Yaskawa INFORM job: CPRINT3D.JBI

/JOB
//NAME CPRINT3D
//POS
///NPOS 981,0,0,0,0,0
///TOOL 9
///POSTYPE PULSE
///PULSE
C00000=20899,58707,-95028,75516,-125126,-84020,0
C00001=20890,61280,-94031,74948,-124335,-84934,0
C00002=20888,61868,-93778,74829,-124164,-85130,0
C00003=21010,62075,-93213,74809,-124380,-84988,0
C00004=21199,62234,-92779,74700,-124608,-84895,0
C00005=21337,62300,-92602,74597,-124739,-84867,0
C00006=38851,62476,-92387,77627,-123060,-84391,0
C00007=39075,62591,-92079,77464,-123273,-84335,0
C00008=39325,62631,-91976,77240,-123458,-84342,0
C00009=39575,62590,-92092,76980,-123593,-84413,0
C00010=39796,62473,-92413,76711,-123659,-84538,0
C00011=39905,62372,-92691,76558,-123665,-84634,0
C00012=51767,54029,-117549,60022,-121835,-93519,0
C00013=51973,53909,-117950,59735,-121747,-93661,0
C00014=52088,53762,-118443,59535,-121588,-93813,0
C00015=52099,53603,-118972,59445,-121375,-93959,0
C00016=52003,53453,-119474,59478,-121135,-94082,0
C00017=51897,53373,-119741,59558,-120988,-94140,0
C00018=29408,51344,-126354,60860,-117429,-95669,0
C00019=29082,51299,-126517,61201,-117262,-95677,0
C00020=28737,51300,-126508,61583,-117162,-95633,0
C00021=28416,51346,-126329,61959,-117138,-95543,0
C00022=28156,51432,-126000,62285,-117193,-95416,0
C00023=28041,51501,-125745,62442,-117261,-95327,0
C00024=20896,61411,-95034,74604,-123854,-85488,0
C00025=20848,61637,-94410,74758,-123981,-85303,0
C00026=20875,61793,-93981,74806,-124105,-85185,0
C00027=23614,61599,-94547,71990,-125641,-85793,0
C00028=23696,61485,-94861,71849,-125604,-85896,0
C00029=23753,61360,-95207,71729,-125543,-86002,0
C00030=23779,61231,-95564,71637,-125461,-86108,0
C00031=23776,61103,-95917,71576,-125361,-86206,0
C00032=23744,60981,-96255,71547,-125249,-86296,0
C00033=23690,60879,-96538,71550,-125138,-86366,0
C00034=23633,60785,-96800,71560,-125033,-86431,0
C00035=23546,60693,-97055,71602,-124911,-86488,0
C00036=23440,60617,-97265,71672,-124790,-86529,0
C00037=23318,60561,-97421,71767,-124676,-86553,0
C00038=23186,60525,-97517,71884,-124572,-86559,0
C00039=23047,60513,-97550,72018,-124482,-86545,0
C00040=22909,60524,-97518,72163,-124411,-86514,0
C00041=22788,60555,-97430,72301,-124363,-86469,0
C00042=22668,60592,-97325,72440,-124321,-86420,0
C00043=22545,60656,-97145,72595,-124297,-86349,0
C00044=22438,60742,-96904,72745,-124300,-86264,0
C00045=22352,60847,-96612,72882,-124326,-86167,0
C00046=22291,60967,-96277,73001,-124380,-86062,0
C00047=22259,61099,-95912,73098,-124457,-85954,0
C00048=22258,61236,-95531,73166,-124557,-85845,0
C00049=22288,61375,-95148,73204,-124675,-85742,0
C00050=22350,61509,-94780,73208,-124810,-85648,0
C00051=22446,61639,-94424,73177,-124961,-85563,0
C00052=22581,61738,-94153,73092,-125115,-85509,0
C00053=22727,61808,-93962,72982,-125256,-85479,0
C00054=22884,61852,-93844,72847,-125383,-85472,0
C00055=23056,61868,-93803,72683,-125500,-85489,0
C00056=23225,61837,-93889,72500,-125581,-85542,0
C00057=23374,61780,-94048,72322,-125629,-85611,0
C00058=23505,61699,-94271,72150,-125649,-85697,0
C00059=23556,61652,-94401,72074,-125645,-85742,0
C00060=23536,61543,-94699,72039,-125552,-85823,0
C00061=23608,61444,-94973,71917,-125521,-85912,0
C00062=23657,61335,-95274,71813,-125468,-86005,0
C00063=23680,61224,-95582,71734,-125397,-86095,0
C00064=23677,61113,-95888,71681,-125311,-86181,0
C00065=23649,61009,-96178,71656,-125214,-86258,0
C00066=23600,60916,-96433,71659,-125115,-86322,0
C00067=23549,60831,-96669,71669,-125019,-86380,0
C00068=23474,60752,-96888,71705,-124914,-86429,0
C00069=23383,60687,-97068,71764,-124812,-86464,0
C00070=23279,60639,-97201,71846,-124713,-86485,0
C00071=23166,60609,-97284,71946,-124625,-86489,0
C00072=23048,60598,-97312,72060,-124548,-86478,0
C00073=22929,60608,-97284,72184,-124486,-86451,0
C00074=22820,60636,-97205,72308,-124443,-86410,0
C00075=22712,60669,-97111,72433,-124405,-86366,0
C00076=22606,60724,-96956,72566,-124385,-86305,0
C00077=22514,60798,-96748,72696,-124386,-86232,0
C00078=22440,60889,-96494,72815,-124410,-86148,0
C00079=22387,60994,-96204,72919,-124456,-86057,0
C00080=22359,61109,-95885,73003,-124524,-85962,0
C00081=22357,61229,-95552,73063,-124611,-85868,0
C00082=22384,61351,-95217,73097,-124716,-85777,0
C00083=22437,61468,-94894,73101,-124833,-85694,0
C00084=22520,61579,-94589,73074,-124964,-85622,0
C00085=22635,61664,-94357,73001,-125095,-85575,0
C00086=22764,61725,-94189,72903,-125219,-85549,0
C00087=22903,61764,-94085,72784,-125332,-85543,0
C00088=23051,61778,-94049,72643,-125431,-85557,0
C00089=23195,61751,-94124,72486,-125499,-85603,0
C00090=23326,61701,-94262,72330,-125542,-85664,0
C00091=23441,61631,-94458,72179,-125559,-85738,0
C00092=23479,61596,-94553,72124,-125557,-85772,0
C00093=23667,61562,-94650,71917,-125644,-85831,0
C00094=22262,61550,-94666,73316,-124787,-85601,0
C00095=22193,61400,-95079,73311,-124636,-85707,0
C00096=22159,61244,-95509,73269,-124503,-85823,0
C00097=22160,61140,-95796,73217,-124427,-85904,0
C00098=22111,61132,-95819,73262,-124393,-85903,0
C00099=21934,61528,-94723,73632,-124571,-85564,0
C00100=22292,61657,-94372,73339,-124881,-85523,0
C00101=22319,61626,-94456,73297,-124876,-85551,0
C00102=22308,61612,-94496,73300,-124859,-85560,0
C00103=29023,52904,-120775,62001,-119581,-94025,0
C00104=29186,52950,-120622,61843,-119699,-94004,0
C00105=29368,52980,-120522,61657,-119804,-94001,0
C00106=29561,52993,-120481,61451,-119889,-94017,0
C00107=29759,52988,-120500,61230,-119951,-94051,0
C00108=29955,52965,-120584,61003,-119987,-94102,0
C00109=30150,52921,-120738,60768,-119993,-94173,0
C00110=30308,52852,-120980,60560,-119950,-94263,0
C00111=30428,52773,-121251,60391,-119880,-94355,0
C00112=30513,52686,-121554,60255,-119785,-94452,0
C00113=30562,52588,-121893,60155,-119660,-94553,0
C00114=30545,52489,-122240,60127,-119511,-94648,0
C00115=30488,52400,-122551,60150,-119363,-94727,0
C00116=30393,52319,-122833,60217,-119215,-94794,0
C00117=30266,52250,-123075,60325,-119072,-94844,0
C00118=30114,52195,-123269,60468,-118942,-94878,0
C00119=29942,52155,-123408,60639,-118828,-94894,0
C00120=29759,52131,-123489,60831,-118734,-94894,0
C00121=29572,52123,-123512,61034,-118664,-94875,0
C00122=29390,52132,-123478,61239,-118619,-94842,0
C00123=29234,52154,-123395,61422,-118601,-94798,0
C00124=29088,52179,-123303,61594,-118591,-94752,0
C00125=28943,52220,-123155,61773,-118602,-94691,0
C00126=28819,52274,-122964,61934,-118638,-94621,0
C00127=28723,52337,-122739,62069,-118695,-94543,0
C00128=28656,52408,-122490,62175,-118773,-94463,0
C00129=28623,52483,-122223,62246,-118868,-94383,0
C00130=28624,52561,-121951,62282,-118976,-94305,0
C00131=28655,52632,-121706,62280,-119085,-94239,0
C00132=28695,52703,-121461,62269,-119195,-94175,0
C00133=28773,52778,-121205,62217,-119324,-94113,0
C00134=28884,52846,-120972,62127,-119455,-94062,0
C00135=28945,52871,-120885,62072,-119510,-94046,0
C00136=29095,52857,-120937,61900,-119543,-94081,0
C00137=29237,52897,-120804,61762,-119645,-94063,0
C00138=29396,52923,-120718,61600,-119736,-94061,0
C00139=29565,52935,-120681,61419,-119811,-94074,0
C00140=29739,52930,-120698,61225,-119865,-94104,0
C00141=29911,52910,-120772,61025,-119896,-94148,0
C00142=30078,52872,-120904,60823,-119901,-94209,0
C00143=30214,52813,-121110,60646,-119864,-94286,0
C00144=30320,52744,-121350,60497,-119802,-94368,0
C00145=30395,52667,-121617,60378,-119718,-94453,0
C00146=30436,52584,-121908,60292,-119612,-94540,0
C00147=30421,52498,-122205,60269,-119485,-94621,0
C00148=30370,52420,-122477,60289,-119355,-94690,0
C00149=30287,52350,-122724,60348,-119225,-94748,0
C00150=30176,52289,-122936,60442,-119101,-94793,0
C00151=30043,52241,-123104,60567,-118987,-94823,0
C00152=29894,52206,-123225,60715,-118888,-94836,0
C00153=29736,52185,-123296,60881,-118807,-94836,0
C00154=29575,52179,-123316,61056,-118746,-94820,0
C00155=29419,52186,-123286,61232,-118707,-94791,0
C00156=29279,52206,-123211,61396,-118691,-94751,0
C00157=29148,52229,-123130,61551,-118681,-94711,0
C00158=29023,52264,-123002,61705,-118691,-94658,0
C00159=28917,52310,-122839,61843,-118722,-94597,0
C00160=28834,52364,-122646,61959,-118771,-94532,0
C00161=28777,52425,-122432,62050,-118838,-94463,0
C00162=28749,52490,-122204,62111,-118918,-94394,0
C00163=28749,52556,-121970,62142,-119011,-94328,0
C00164=28777,52620,-121750,62141,-119109,-94268,0
C00165=28812,52684,-121530,62131,-119209,-94210,0
C00166=28879,52748,-121308,62087,-119319,-94157,0
C00167=28975,52807,-121107,62009,-119433,-94113,0
C00168=29017,52824,-121047,61971,-119472,-94101,0
C00169=29079,52934,-120675,61954,-119641,-94004,0
C00170=48817,53183,-120295,62872,-119678,-93851,0
C00171=48657,53224,-120148,63068,-119677,-93787,0
C00172=48515,53282,-119949,63250,-119702,-93711,0
C00173=48399,53354,-119702,63411,-119755,-93624,0
C00174=48315,53438,-119417,63544,-119832,-93531,0
C00175=48265,53531,-119102,63641,-119933,-93435,0
C00176=48255,53630,-118772,63700,-120053,-93339,0
C00177=48286,53736,-118420,63715,-120197,-93244,0
C00178=48378,53834,-118099,63660,-120352,-93165,0
C00179=48500,53917,-117828,63567,-120500,-93106,0
C00180=48649,53987,-117600,63436,-120643,-93063,0
C00181=48830,54045,-117416,63265,-120782,-93038,0
C00182=49033,54072,-117332,63055,-120891,-93043,0
C00183=49230,54078,-117320,62842,-120972,-93069,0
C00184=49421,54063,-117371,62626,-121026,-93112,0
C00185=49598,54031,-117484,62415,-121050,-93170,0
C00186=49755,53982,-117647,62219,-121046,-93239,0
C00187=49891,53919,-117860,62040,-121015,-93318,0
C00188=49996,53845,-118106,61888,-120959,-93403,0
C00189=50069,53764,-118377,61769,-120880,-93490,0
C00190=50108,53679,-118661,61685,-120783,-93574,0
C00191=50111,53600,-118923,61643,-120681,-93648,0
C00192=50107,53526,-119172,61613,-120581,-93717,0
C00193=50069,53445,-119442,61616,-120461,-93787,0
C00194=50000,53370,-119695,61656,-120336,-93848,0
C00195=49902,53303,-119919,61733,-120212,-93897,0
C00196=49778,53246,-120107,61842,-120094,-93933,0
C00197=49634,53202,-120252,61980,-119986,-93953,0
C00198=49475,53172,-120349,62141,-119891,-93958,0
C00199=49321,53160,-120388,62305,-119821,-93947,0
C00200=49166,53151,-120413,62473,-119756,-93933,0
C00201=48989,53158,-120383,62670,-119705,-93900,0
C00202=48915,53169,-120345,62757,-119694,-93879,0
C00203=48866,53237,-120111,62843,-119767,-93806,0
C00204=48727,53273,-119983,63013,-119766,-93750,0
C00205=48605,53324,-119811,63171,-119788,-93684,0
C00206=48504,53387,-119595,63312,-119833,-93609,0
C00207=48429,53460,-119346,63428,-119901,-93527,0
C00208=48386,53542,-119071,63514,-119989,-93443,0
C00209=48376,53628,-118781,63566,-120095,-93359,0
C00210=48402,53719,-118480,63580,-120219,-93277,0
C00211=48481,53803,-118204,63533,-120352,-93210,0
C00212=48588,53876,-117964,63450,-120483,-93157,0
C00213=48720,53938,-117764,63335,-120608,-93119,0
C00214=48875,53987,-117607,63188,-120728,-93097,0
C00215=49050,54010,-117534,63008,-120821,-93103,0
C00216=49223,54015,-117524,62820,-120891,-93125,0
C00217=49390,54003,-117569,62631,-120938,-93163,0
C00218=49546,53975,-117667,62446,-120959,-93213,0
C00219=49683,53932,-117810,62275,-120956,-93274,0
C00220=49800,53877,-117994,62119,-120929,-93343,0
C00221=49891,53814,-118208,61988,-120880,-93416,0
C00222=49954,53744,-118442,61886,-120812,-93491,0
C00223=49987,53670,-118686,61814,-120728,-93564,0
C00224=49990,53600,-118923,61777,-120637,-93630,0
C00225=49986,53533,-119147,61750,-120548,-93693,0
C00226=49953,53463,-119378,61753,-120444,-93753,0
C00227=49894,53399,-119594,61787,-120337,-93805,0
C00228=49809,53341,-119787,61853,-120232,-93847,0
C00229=49704,53292,-119948,61946,-120130,-93877,0
C00230=49580,53255,-120072,62064,-120037,-93895,0
C00231=49444,53229,-120155,62202,-119957,-93899,0
C00232=49306,53218,-120190,62350,-119894,-93889,0
C00233=49166,53210,-120212,62500,-119835,-93876,0
C00234=49015,53216,-120187,62670,-119790,-93848,0
C00235=48964,53223,-120161,62728,-119782,-93834,0
C00236=48738,53191,-120265,62963,-119662,-93832,0
C00237=49561,53062,-120729,61994,-119772,-94078,0
C00238=30717,52351,-122728,59873,-119365,-94808,0
C00239=30793,52470,-122309,59844,-119565,-94702,0
C00240=30814,52599,-121862,59881,-119758,-94580,0
C00241=30750,52724,-121427,60011,-119918,-94449,0
C00242=30644,52832,-121052,60179,-120036,-94330,0
C00243=30495,52929,-120716,60390,-120122,-94216,0
C00244=30292,53019,-120407,60657,-120176,-94101,0
C00245=30041,53076,-120209,60960,-120168,-94009,0
C00246=29799,53105,-120105,61241,-120124,-93946,0
C00247=29553,53111,-120080,61515,-120045,-93903,0
C00248=29312,53094,-120133,61773,-119939,-93884,0
C00249=29084,53056,-120258,62005,-119808,-93887,0
C00250=28879,52998,-120450,62204,-119658,-93913,0
C00251=28702,52924,-120699,62363,-119497,-93960,0
C00252=28562,52837,-120996,62478,-119331,-94024,0
C00253=28461,52742,-121323,62544,-119166,-94104,0
C00254=28412,52657,-121616,62558,-119034,-94181,0
C00255=28369,52561,-121948,62562,-118889,-94270,0
C00256=22538,60451,-97717,72502,-124139,-86510,0
C00257=22723,60394,-97878,72288,-124203,-86586,0
C00258=22869,60358,-97983,72122,-124259,-86639,0
C00259=23047,60344,-98024,71935,-124352,-86680,0
C00260=23226,60359,-97982,71762,-124467,-86696,0
C00261=23396,60404,-97858,71611,-124601,-86690,0
C00262=23553,60477,-97658,71487,-124747,-86659,0
C00263=23690,60574,-97388,71397,-124902,-86606,0
C00264=23801,60692,-97061,71343,-125058,-86532,0
C00265=23870,60805,-96746,71330,-125187,-86456,0
C00266=23934,60927,-96407,71327,-125319,-86371,0
C00267=23974,61083,-95975,71365,-125463,-86256,0
C00268=23978,61246,-95525,71444,-125590,-86130,0
C00269=23944,61410,-95073,71561,-125695,-85997,0
C00270=23873,61568,-94637,71714,-125772,-85863,0
C00271=23768,61711,-94241,71892,-125816,-85733,0
C00272=23632,61836,-93895,72092,-125828,-85613,0
C00273=23468,61937,-93617,72307,-125803,-85506,0
C00274=23380,61971,-93523,72413,-125774,-85465,0
C00275=38247,60799,-96991,77469,-121636,-85632,0
C00276=38229,60634,-97453,77414,-121520,-85763,0
C00277=38224,60505,-97812,77364,-121434,-85867,0
C00278=38252,60358,-98224,77272,-121355,-85990,0
C00279=38315,60220,-98614,77149,-121301,-86112,0
C00280=38410,60095,-98966,77001,-121276,-86226,0
C00281=38534,59989,-99267,76833,-121277,-86331,0
C00282=38681,59906,-99506,76650,-121307,-86420,0
C00283=38846,59848,-99673,76460,-121365,-86492,0
C00284=38995,59822,-99749,76300,-121432,-86534,0
C00285=39152,59803,-99808,76134,-121511,-86573,0
C00286=39341,59810,-99789,75949,-121624,-86594,0
C00287=39527,59849,-99684,75780,-121759,-86589,0
C00288=39702,59918,-99492,75635,-121908,-86558,0
C00289=39859,60016,-99219,75522,-122067,-86502,0
C00290=39990,60139,-98875,75446,-122229,-86422,0
C00291=40090,60284,-98470,75413,-122389,-86319,0
C00292=40154,60445,-98019,75422,-122538,-86199,0
C00293=40165,60527,-97789,75448,-122601,-86135,0
C00294=49264,54203,-116909,62865,-121141,-92959,0
C00295=49001,54196,-116927,63150,-121033,-92924,0
C00296=48740,54161,-117035,63420,-120891,-92916,0
C00297=48507,54087,-117270,63639,-120712,-92949,0
C00298=48323,53999,-117551,63799,-120536,-93002,0
C00299=48172,53896,-117887,63915,-120353,-93075,0
C00300=48053,53770,-118301,63986,-120153,-93176,0
C00301=48012,53634,-118754,63967,-119970,-93300,0
C00302=48024,53511,-119164,63896,-119820,-93419,0
C00303=48085,53395,-119556,63776,-119695,-93540,0
C00304=48190,53290,-119913,63611,-119597,-93656,0
C00305=48335,53199,-120225,63409,-119532,-93765,0
C00306=48514,53127,-120476,63179,-119500,-93862,0
C00307=48718,53074,-120661,62930,-119501,-93942,0
C00308=48938,53043,-120775,62673,-119534,-94005,0
C00309=49164,53034,-120813,62419,-119600,-94047,0
C00310=49352,53044,-120783,62217,-119677,-94064,0
C00311=49459,53053,-120756,62103,-119725,-94071,0
C00312=50348,53502,-119261,61335,-120633,-93777,0
C00313=50354,53603,-118923,61377,-120769,-93684,0
C00314=50347,53723,-118523,61442,-120924,-93571,0
C00315=50567,53630,-118838,61154,-120880,-93692,0
C00316=50415,53540,-119133,61280,-120708,-93751,0
C00317=29384,52018,-123887,61194,-118449,-94958,0
C00318=29114,51954,-124111,61462,-118270,-94987,0
C00319=28946,52085,-123636,61708,-118408,-94829,0
C00320=29144,52051,-123761,61474,-118423,-94890,0
C00321=29282,52032,-123833,61312,-118438,-94929,0
C00322=28535,52391,-122546,62301,-118709,-94463,0
C00323=28611,52310,-122832,62180,-118620,-94556,0
C00324=28721,52238,-123089,62026,-118555,-94643,0
C00325=28862,52177,-123307,61842,-118514,-94724,0
C00326=29028,52130,-123477,61638,-118500,-94795,0
C00327=29189,52103,-123578,61448,-118511,-94844,0
C00328=29361,52078,-123669,61246,-118531,-94892,0
C00329=29569,52068,-123709,61012,-118583,-94931,0
C00330=29760,52076,-123686,60804,-118654,-94950,0
C00331=29778,52051,-123776,60773,-118623,-94977,0
C00332=29062,51880,-124374,61486,-118145,-95056,0
C00333=22333,60653,-97151,72807,-124171,-86316,0
C00334=22373,60676,-97086,72778,-124212,-86305,0
C00335=22483,60588,-97333,72624,-124210,-86392,0
C00336=22623,60515,-97539,72447,-124238,-86474,0
C00337=22755,60475,-97654,72294,-124283,-86527,0
C00338=22889,60441,-97751,72142,-124335,-86576,0
C00339=23047,60428,-97787,71976,-124417,-86612,0
C00340=23206,60442,-97750,71823,-124519,-86628,0
C00341=23357,60482,-97640,71689,-124639,-86622,0
C00342=23497,60547,-97462,71580,-124768,-86594,0
C00343=23618,60633,-97222,71500,-124906,-86547,0
C00344=23717,60738,-96931,71452,-125045,-86481,0
C00345=23780,60842,-96642,71440,-125163,-86411,0
C00346=23839,60954,-96331,71437,-125284,-86333,0
C00347=23875,61093,-95946,71470,-125412,-86231,0
C00348=23878,61238,-95544,71540,-125526,-86119,0
C00349=23848,61385,-95140,71645,-125619,-86000,0
C00350=23785,61526,-94749,71781,-125688,-85879,0
C00351=23691,61655,-94394,71941,-125728,-85763,0
C00352=23568,61768,-94083,72121,-125738,-85655,0
C00353=23421,61858,-93832,72314,-125716,-85559,0
C00354=23254,61923,-93655,72514,-125661,-85481,0
C00355=23157,61940,-93605,72620,-125614,-85450,0
C00356=23152,61980,-93497,72644,-125641,-85419,0
C00357=38423,61024,-96369,77395,-121886,-85476,0
C00358=38460,60998,-96443,77347,-121892,-85503,0
C00359=38389,60883,-96762,77366,-121775,-85585,0
C00360=38342,60748,-97137,77353,-121660,-85687,0
C00361=38330,60629,-97468,77313,-121576,-85781,0
C00362=38325,60511,-97797,77267,-121498,-85876,0
C00363=38351,60381,-98163,77184,-121428,-85986,0
C00364=38407,60258,-98510,77075,-121381,-86094,0
C00365=38491,60147,-98823,76943,-121358,-86196,0
C00366=38601,60052,-99091,76793,-121359,-86289,0
C00367=38732,59978,-99303,76631,-121386,-86368,0
C00368=38879,59927,-99451,76462,-121437,-86431,0
C00369=39015,59903,-99521,76316,-121499,-86471,0
C00370=39159,59885,-99575,76164,-121570,-86506,0
C00371=39327,59892,-99558,76000,-121673,-86525,0
C00372=39493,59926,-99464,75849,-121792,-86521,0
C00373=39649,59988,-99292,75720,-121927,-86493,0
C00374=39789,60076,-99048,75619,-122068,-86443,0
C00375=39907,60187,-98738,75551,-122214,-86370,0
C00376=39997,60317,-98375,75520,-122356,-86279,0
C00377=40055,60462,-97968,75529,-122491,-86170,0
C00378=40077,60617,-97535,75578,-122610,-86048,0
C00379=40068,60704,-97293,75626,-122665,-85978,0
C00380=40109,60718,-97253,75592,-122700,-85972,0
C00381=49614,54127,-117170,62444,-121176,-93084,0
C00382=49583,54100,-117256,62465,-121131,-93104,0
C00383=49451,54124,-117174,62622,-121113,-93061,0
C00384=49238,54140,-117115,62864,-121052,-93013,0
C00385=49017,54134,-117130,63103,-120962,-92984,0
C00386=48785,54103,-117225,63343,-120836,-92977,0
C00387=48578,54037,-117436,63538,-120679,-93006,0
C00388=48411,53958,-117690,63683,-120519,-93054,0
C00389=48275,53865,-117993,63788,-120353,-93121,0
C00390=48169,53753,-118361,63851,-120175,-93210,0
C00391=48133,53632,-118763,63833,-120011,-93320,0
C00392=48145,53521,-119133,63769,-119876,-93427,0
C00393=48200,53416,-119486,63659,-119763,-93536,0
C00394=48295,53322,-119808,63511,-119675,-93641,0
C00395=48425,53241,-120087,63329,-119617,-93738,0
C00396=48586,53176,-120312,63123,-119588,-93824,0
C00397=48767,53128,-120479,62901,-119589,-93897,0
C00398=48964,53100,-120579,62671,-119619,-93953,0
C00399=49165,53092,-120613,62446,-119678,-93990,0
C00400=49337,53102,-120585,62261,-119749,-94006,0
C00401=49506,53116,-120542,62080,-119826,-94017,0
C00402=49688,53150,-120433,61895,-119934,-94012,0
C00403=49853,53200,-120267,61737,-120058,-93988,0
C00404=49994,53264,-120051,61612,-120192,-93947,0
C00405=50106,53341,-119794,61525,-120335,-93891,0
C00406=50185,53427,-119505,61479,-120477,-93822,0
C00407=50228,53519,-119197,61476,-120614,-93742,0
C00408=50233,53601,-118924,61510,-120725,-93666,0
C00409=50228,53688,-118635,61557,-120837,-93585,0
C00410=50183,53785,-118311,61653,-120947,-93488,0
C00411=50109,53868,-118034,61775,-121028,-93400,0
C00412=50155,53886,-117976,61733,-121068,-93390,0
C00413=50738,53638,-118816,60970,-120951,-93711,0
C00414=30446,52217,-123195,60111,-119081,-94902,0
C00415=30405,52238,-123122,60165,-119098,-94876,0
C00416=30499,52289,-122941,60085,-119204,-94838,0
C00417=30605,52380,-122624,60010,-119372,-94764,0
C00418=30669,52480,-122275,59986,-119539,-94675,0
C00419=30688,52594,-121878,60018,-119710,-94567,0
C00420=30632,52705,-121490,60133,-119851,-94451,0
C00421=30536,52803,-121152,60285,-119958,-94343,0
C00422=30402,52890,-120849,60475,-120036,-94239,0
C00423=30221,52970,-120573,60712,-120084,-94137,0
C00424=29998,53020,-120397,60982,-120078,-94055,0
C00425=29779,53046,-120303,61235,-120037,-93998,0
C00426=29557,53052,-120281,61483,-119967,-93960,0
C00427=29339,53037,-120327,61715,-119872,-93943,0
C00428=29135,53003,-120441,61924,-119754,-93946,0
C00429=28951,52951,-120613,62103,-119620,-93969,0
C00430=28793,52885,-120836,62246,-119475,-94011,0
C00431=28667,52807,-121100,62348,-119327,-94069,0
C00432=28578,52722,-121392,62407,-119180,-94140,0
C00433=28534,52644,-121661,62419,-119059,-94210,0
C00434=28499,52566,-121931,62422,-118941,-94283,0
C00435=28498,52477,-122241,62382,-118817,-94372,0
C00436=28515,52437,-122384,62344,-118766,-94415,0
C00437=38572,60199,-98679,76886,-121439,-86166,0
C00438=38498,60295,-98405,77002,-121460,-86076,0
C00439=38449,60403,-98102,77097,-121501,-85981,0
C00440=38426,60518,-97781,77170,-121562,-85885,0
C00441=38430,60625,-97482,77212,-121635,-85799,0
C00442=38441,60733,-97181,77249,-121711,-85714,0
C00443=38482,60851,-96852,77260,-121812,-85624,0
C00444=38551,60963,-96542,77242,-121925,-85544,0
C00445=38646,61063,-96265,77193,-122047,-85477,0
C00446=38763,61148,-96032,77115,-122174,-85427,0
C00447=38900,61213,-95856,77010,-122298,-85396,0
C00448=39051,61254,-95745,76880,-122417,-85385,0
C00449=39211,61269,-95707,76730,-122524,-85397,0
C00450=39373,61256,-95745,76565,-122615,-85432,0
C00451=39540,61213,-95868,76380,-122688,-85491,0
C00452=39685,61128,-96106,76199,-122721,-85580,0
C00453=39803,61026,-96392,76036,-122724,-85680,0
C00454=39895,60906,-96726,75890,-122699,-85790,0
C00455=39961,60767,-97115,75761,-122645,-85911,0
C00456=39976,60618,-97531,75679,-122552,-86033,0
C00457=39956,60480,-97917,75636,-122445,-86141,0
C00458=39904,60350,-98279,75628,-122325,-86237,0
C00459=39824,60235,-98602,75656,-122199,-86319,0
C00460=39720,60136,-98877,75716,-122070,-86383,0
C00461=39596,60059,-99092,75805,-121944,-86428,0
C00462=39458,60004,-99244,75918,-121827,-86452,0
C00463=39312,59974,-99327,76050,-121721,-86456,0
C00464=39165,59968,-99341,76194,-121631,-86439,0
C00465=39034,59984,-99292,76332,-121566,-86407,0
C00466=38911,60006,-99229,76465,-121509,-86372,0
C00467=38783,60051,-99099,76612,-121465,-86316,0
C00468=38668,60116,-98913,76754,-121440,-86247,0
C00469=38631,60148,-98822,76806,-121440,-86215,0
C00470=38653,60251,-98534,76829,-121521,-86135,0
C00471=38589,60334,-98300,76928,-121538,-86058,0
C00472=38547,60426,-98040,77010,-121574,-85977,0
C00473=38527,60524,-97765,77073,-121627,-85895,0
C00474=38530,60621,-97495,77111,-121692,-85817,0
C00475=38540,60717,-97225,77144,-121760,-85740,0
C00476=38575,60819,-96942,77155,-121847,-85663,0
C00477=38635,60916,-96674,77139,-121946,-85594,0
C00478=38717,61003,-96434,77097,-122052,-85536,0
C00479=38819,61076,-96232,77029,-122161,-85492,0
C00480=38938,61133,-96078,76937,-122270,-85465,0
C00481=39070,61169,-95981,76823,-122374,-85456,0
C00482=39210,61182,-95948,76691,-122468,-85466,0
C00483=39353,61170,-95982,76545,-122547,-85496,0
C00484=39497,61133,-96087,76387,-122610,-85548,0
C00485=39621,61061,-96290,76232,-122638,-85624,0
C00486=39725,60971,-96543,76089,-122640,-85712,0
C00487=39806,60865,-96838,75960,-122618,-85809,0
C00488=39862,60746,-97171,75850,-122571,-85913,0
C00489=39875,60619,-97527,75780,-122492,-86016,0
C00490=39857,60498,-97865,75742,-122399,-86112,0
C00491=39811,60384,-98182,75736,-122294,-86196,0
C00492=39741,60283,-98465,75760,-122184,-86268,0
C00493=39650,60197,-98704,75812,-122071,-86324,0
C00494=39543,60130,-98892,75890,-121962,-86363,0
C00495=39423,60082,-99023,75988,-121860,-86384,0
C00496=39298,60056,-99095,76101,-121769,-86387,0
C00497=39171,60051,-99107,76225,-121691,-86373,0
C00498=39054,60065,-99063,76349,-121632,-86343,0
C00499=38943,60085,-99006,76467,-121581,-86312,0
C00500=38833,60124,-98894,76594,-121543,-86264,0
C00501=38735,60180,-98735,76716,-121523,-86204,0
C00502=38711,60200,-98677,76748,-121522,-86184,0
C00503=38534,60236,-98572,76940,-121442,-86129,0
C00504=38895,61347,-95485,77074,-122382,-85288,0
C00505=39275,61614,-94754,76823,-122787,-85132,0
C00506=39516,61348,-95493,76466,-122763,-85379,0
C00507=39491,61316,-95581,76476,-122726,-85401,0
C00508=39393,61342,-95508,76585,-122683,-85366,0
C00509=39211,61356,-95465,76770,-122580,-85327,0
C00510=39032,61339,-95508,76938,-122460,-85314,0
C00511=38951,61317,-95567,77007,-122397,-85320,0
C00512=39291,61738,-94413,76864,-122876,-85036,0
C00513=50908,53647,-118792,60786,-121022,-93730,0
C00514=29010,51808,-124637,61511,-118019,-95125,0
C00515=21806,61577,-94585,73782,-124528,-85505,0
C00516=39226,61692,-94540,76906,-122806,-85064,0
C00517=39307,61863,-94071,76905,-122965,-84941,0
C00518=51079,53656,-118768,60601,-121093,-93748,0
C00519=28958,51735,-124901,61536,-117895,-95194,0
C00520=21679,61627,-94447,73933,-124485,-85445,0
C00521=39243,61816,-94198,76947,-122895,-84968,0
C00522=39528,61412,-95316,76484,-122811,-85331,0
C00523=39327,61486,-95109,76714,-122737,-85242,0
C00524=39050,61399,-95344,76947,-122510,-85269,0
C00525=38862,61308,-95592,77089,-122336,-85314,0
C00526=38788,61264,-95710,77143,-122262,-85337,0
C00527=38713,61221,-95828,77198,-122189,-85361,0
C00528=38570,61122,-96101,77293,-122038,-85420,0
C00529=38508,61069,-96248,77331,-121967,-85453,0
C00530=38476,61042,-96320,77350,-121930,-85470,0
C00531=38345,60913,-96678,77422,-121768,-85555,0
C00532=38304,60868,-96802,77442,-121714,-85585,0
C00533=38315,60856,-96835,77426,-121714,-85596,0
C00534=38326,60906,-96697,77437,-121752,-85558,0
C00535=38315,60856,-96835,77426,-121714,-85596,0
C00536=38304,60806,-96974,77416,-121675,-85635,0
C00537=38073,60621,-97486,77562,-121417,-85752,0
C00538=38183,60609,-97521,77449,-121475,-85777,0
C00539=38179,60524,-97759,77416,-121419,-85845,0
C00540=37959,60547,-97689,77642,-121301,-85795,0
C00541=37845,60475,-97890,77723,-121186,-85838,0
C00542=38188,60438,-98000,77370,-121368,-85916,0
C00543=38205,60351,-98243,77315,-121322,-85989,0
C00544=37731,60402,-98091,77805,-121073,-85881,0
C00545=37616,60330,-98291,77887,-120958,-85924,0
C00546=38240,60263,-98491,77243,-121285,-86066,0
C00547=38280,60175,-98740,77165,-121252,-86143,0
C00548=37501,60259,-98490,77970,-120844,-85967,0
C00549=37386,60187,-98688,78054,-120730,-86009,0
C00550=38350,60084,-98997,77057,-121232,-86228,0
C00551=38385,60039,-99126,77002,-121223,-86269,0
C00552=38439,59991,-99259,76927,-121224,-86316,0
C00553=37271,60116,-98885,78138,-120617,-86051,0
C00554=37155,60046,-99081,78223,-120503,-86093,0
C00555=38566,59896,-99531,76760,-121234,-86412,0
C00556=38686,59828,-99725,76611,-121258,-86485,0
C00557=38790,59792,-99830,76492,-121293,-86529,0
C00558=37038,59976,-99277,78308,-120390,-86135,0
C00559=40365,60246,-98581,75121,-122522,-86392,0
C00560=40131,60263,-98528,75362,-122398,-86343,0
C00561=40128,60255,-98552,75362,-122390,-86349,0
C00562=40079,60183,-98752,75378,-122312,-86399,0
C00563=40456,60156,-98837,74988,-122511,-86479,0
C00564=40548,60066,-99091,74855,-122500,-86565,0
C00565=40024,60104,-98974,75397,-122224,-86455,0
C00566=40018,60096,-98997,75399,-122215,-86461,0
C00567=39944,60027,-99190,75441,-122124,-86506,0
C00568=40640,59977,-99345,74721,-122490,-86652,0
C00569=40732,59888,-99598,74587,-122478,-86738,0
C00570=39858,59950,-99404,75494,-122021,-86555,0
C00571=39739,59877,-99610,75580,-121900,-86598,0
C00572=40825,59799,-99850,74453,-122468,-86825,0
C00573=40918,59711,-100102,74319,-122456,-86911,0
C00574=39583,59806,-99805,75705,-121761,-86633,0
C00575=39506,59776,-99889,75768,-121696,-86646,0
C00576=39347,59743,-99979,75913,-121582,-86649,0
C00577=41011,59624,-100352,74184,-122445,-86996,0
C00578=41105,59537,-100602,74049,-122432,-87082,0
C00579=36922,59906,-99471,78394,-120276,-86177,0
C00580=36805,59837,-99665,78481,-120164,-86219,0
C00581=41199,59450,-100850,73913,-122421,-87168,0
C00582=41294,59364,-101098,73777,-122409,-87253,0
C00583=36687,59768,-99858,78569,-120051,-86261,0
C00584=36569,59699,-100051,78657,-119940,-86302,0
C00585=41389,59278,-101345,73641,-122397,-87338,0
C00586=41484,59193,-101591,73505,-122384,-87422,0
C00587=36452,59631,-100242,78746,-119827,-86343,0
C00588=36333,59563,-100432,78835,-119716,-86384,0
C00589=41579,59108,-101837,73368,-122371,-87507,0
C00590=41675,59023,-102081,73231,-122359,-87592,0
C00591=36214,59495,-100622,78925,-119604,-86425,0
C00592=36095,59428,-100811,79016,-119493,-86466,0
C00593=41772,58939,-102325,73093,-122346,-87677,0
C00594=41868,58855,-102568,72955,-122333,-87761,0
C00595=35976,59362,-100999,79108,-119381,-86507,0
C00596=35856,59295,-101186,79200,-119271,-86547,0
C00597=41965,58772,-102810,72817,-122321,-87844,0
C00598=42063,58689,-103051,72678,-122307,-87928,0
C00599=35736,59229,-101372,79292,-119161,-86587,0
C00600=35616,59164,-101558,79386,-119050,-86628,0
C00601=42161,58607,-103291,72539,-122293,-88012,0
C00602=42259,58525,-103531,72400,-122279,-88096,0
C00603=35495,59098,-101742,79480,-118940,-86668,0
C00604=35374,59033,-101926,79574,-118830,-86708,0
C00605=42357,58443,-103770,72260,-122266,-88179,0
C00606=42456,58362,-104007,72120,-122252,-88262,0
C00607=35253,58969,-102109,79670,-118720,-86748,0
C00608=35131,58905,-102291,79766,-118611,-86788,0
C00609=42555,58281,-104245,71980,-122238,-88345,0
C00610=42655,58201,-104481,71839,-122224,-88427,0
C00611=35009,58841,-102473,79862,-118502,-86827,0
C00612=34886,58777,-102653,79959,-118393,-86867,0
C00613=42755,58121,-104717,71698,-122209,-88510,0
C00614=42856,58041,-104951,71557,-122194,-88593,0
C00615=34763,58714,-102833,80057,-118284,-86905,0
C00616=34640,58651,-103012,80156,-118176,-86945,0
C00617=42956,57962,-105185,71415,-122181,-88675,0
C00618=43058,57884,-105418,71273,-122166,-88757,0
C00619=34517,58589,-103190,80255,-118068,-86984,0
C00620=34393,58527,-103367,80354,-117960,-87023,0
C00621=43159,57805,-105651,71130,-122149,-88839,0
C00622=43261,57727,-105882,70987,-122135,-88921,0
C00623=34269,58465,-103544,80455,-117852,-87061,0
C00624=34144,58404,-103719,80556,-117744,-87100,0
C00625=43364,57650,-106113,70844,-122120,-89002,0
C00626=43466,57573,-106343,70700,-122104,-89084,0
C00627=34019,58343,-103894,80658,-117637,-87138,0
C00628=33894,58282,-104068,80760,-117530,-87176,0
C00629=43570,57496,-106572,70556,-122087,-89165,0
C00630=43673,57420,-106801,70412,-122072,-89246,0
C00631=33768,58222,-104241,80863,-117423,-87215,0
C00632=33642,58162,-104414,80966,-117316,-87253,0
C00633=43777,57344,-107029,70267,-122056,-89327,0
C00634=43882,57268,-107256,70121,-122039,-89407,0
C00635=33516,58102,-104585,81070,-117209,-87291,0
C00636=33389,58043,-104756,81175,-117104,-87328,0
C00637=43986,57193,-107482,69976,-122023,-89488,0
C00638=44091,57119,-107707,69830,-122007,-89568,0
C00639=33262,57984,-104926,81281,-116998,-87366,0
C00640=33135,57926,-105095,81387,-116892,-87404,0
C00641=44197,57044,-107932,69684,-121990,-89649,0
C00642=44303,56970,-108156,69537,-121973,-89728,0
C00643=33007,57867,-105264,81493,-116786,-87441,0
C00644=32879,57810,-105431,81601,-116682,-87479,0
C00645=44410,56897,-108379,69390,-121955,-89808,0
C00646=44516,56824,-108601,69242,-121938,-89888,0
C00647=32751,57752,-105598,81708,-116577,-87516,0
C00648=32622,57695,-105764,81817,-116472,-87552,0
C00649=44623,56751,-108823,69094,-121921,-89967,0
C00650=44731,56679,-109044,68946,-121904,-90047,0
C00651=32493,57638,-105930,81926,-116367,-87590,0
C00652=32363,57581,-106094,82036,-116264,-87626,0
C00653=44839,56607,-109264,68797,-121885,-90126,0
C00654=44948,56535,-109483,68648,-121868,-90205,0
C00655=32233,57525,-106258,82146,-116159,-87663,0
C00656=32103,57469,-106420,82257,-116056,-87699,0
C00657=45057,56464,-109702,68498,-121850,-90284,0
C00658=45166,56393,-109919,68348,-121831,-90363,0
C00659=31973,57414,-106582,82369,-115952,-87736,0
C00660=31842,57359,-106744,82481,-115849,-87772,0
C00661=45276,56323,-110137,68198,-121813,-90442,0
C00662=45386,56253,-110353,68047,-121793,-90520,0
C00663=31711,57304,-106904,82594,-115745,-87808,0
C00664=31579,57249,-107064,82707,-115643,-87844,0
C00665=45496,56183,-110569,67896,-121775,-90598,0
C00666=45607,56114,-110784,67745,-121755,-90676,0
C00667=31447,57195,-107223,82821,-115541,-87880,0
C00668=31315,57141,-107381,82936,-115438,-87916,0
C00669=45719,56045,-110998,67593,-121737,-90754,0
C00670=45831,55976,-111211,67440,-121717,-90831,0
C00671=31182,57088,-107538,83051,-115336,-87951,0
C00672=31049,57035,-107694,83167,-115234,-87987,0
C00673=45943,55908,-111424,67287,-121698,-90909,0
C00674=46056,55840,-111636,67134,-121678,-90986,0
C00675=30916,56982,-107850,83283,-115133,-88022,0
C00676=30782,56929,-108005,83400,-115032,-88057,0
C00677=46169,55773,-111847,66980,-121658,-91064,0
C00678=46282,55706,-112057,66826,-121638,-91140,0
C00679=30648,56877,-108159,83518,-114930,-88093,0
C00680=30514,56825,-108313,83636,-114829,-88127,0
C00681=46396,55639,-112267,66672,-121617,-91217,0
C00682=46511,55573,-112476,66517,-121597,-91294,0
C00683=30379,56774,-108465,83755,-114728,-88162,0
C00684=30244,56722,-108617,83875,-114628,-88197,0
C00685=46626,55507,-112685,66361,-121576,-91371,0
C00686=46741,55442,-112892,66206,-121555,-91447,0
C00687=30108,56671,-108768,83995,-114528,-88232,0
C00688=29972,56621,-108918,84115,-114428,-88266,0
C00689=46857,55376,-113099,66050,-121535,-91523,0
C00690=46973,55312,-113305,65893,-121513,-91599,0
C00691=29836,56571,-109068,84237,-114328,-88300,0
C00692=29700,56521,-109216,84358,-114229,-88335,0
C00693=47090,55247,-113511,65736,-121492,-91675,0
C00694=47207,55183,-113715,65578,-121470,-91750,0
C00695=29563,56471,-109364,84481,-114129,-88369,0
C00696=29425,56422,-109511,84604,-114030,-88403,0
C00697=47325,55119,-113919,65421,-121449,-91825,0
C00698=47443,55056,-114122,65262,-121427,-91901,0
C00699=29288,56373,-109657,84728,-113932,-88437,0
C00700=29150,56324,-109803,84852,-113833,-88470,0
C00701=47561,54993,-114325,65103,-121405,-91976,0
C00702=47680,54931,-114527,64944,-121382,-92051,0
C00703=29012,56276,-109947,84977,-113735,-88504,0
C00704=28873,56228,-110091,85102,-113637,-88538,0
C00705=47800,54868,-114728,64784,-121360,-92125,0
C00706=47920,54806,-114928,64624,-121337,-92200,0
C00707=28734,56180,-110234,85228,-113539,-88571,0
C00708=28594,56133,-110377,85354,-113441,-88604,0
C00709=48040,54745,-115128,64464,-121314,-92275,0
C00710=48161,54684,-115327,64303,-121291,-92349,0
C00711=28455,56086,-110518,85482,-113344,-88637,0
C00712=28315,56039,-110659,85609,-113247,-88671,0
C00713=48282,54623,-115525,64141,-121268,-92423,0
C00714=48404,54563,-115722,63979,-121245,-92497,0
C00715=28174,55992,-110799,85738,-113150,-88703,0
C00716=24109,62203,-92899,71803,-126391,-85416,0
C00717=48526,54503,-115920,63817,-121221,-92571,0
C00718=48649,54443,-116115,63654,-121198,-92644,0
C00719=23982,62151,-93038,71903,-126275,-85433,0
C00720=23856,62100,-93176,72004,-126160,-85449,0
C00721=48772,54383,-116311,63491,-121174,-92717,0
C00722=48895,54324,-116505,63328,-121150,-92790,0
C00723=23729,62049,-93314,72104,-126044,-85466,0
C00724=23601,61999,-93450,72206,-125929,-85483,0
C00725=49001,54265,-116701,63183,-121118,-92861,0
C00726=49004,54254,-116737,63175,-121105,-92872,0
C00727=48760,54221,-116838,63426,-120972,-92864,0
C00728=48666,54191,-116933,63514,-120900,-92877,0
C00729=23711,61863,-93824,72027,-125896,-85606,0
C00730=23795,61785,-94038,71903,-125889,-85681,0
C00731=23842,61720,-94218,71822,-125868,-85740,0
C00732=48468,54122,-117153,63699,-120741,-92910,0
C00733=48328,54056,-117367,63821,-120607,-92951,0
C00734=23924,61596,-94560,71677,-125824,-85850,0
C00735=23975,61483,-94870,71568,-125769,-85946,0
C00736=48225,53991,-117577,63902,-120489,-92995,0
C00737=48133,53926,-117786,63973,-120375,-93042,0
C00738=24004,61379,-95159,71485,-125707,-86032,0
C00739=24025,61277,-95439,71412,-125642,-86114,0
C00740=48073,53863,-117993,64008,-120276,-93092,0
C00741=48013,53800,-118200,64044,-120176,-93142,0
C00742=24025,61184,-95697,71365,-125571,-86186,0
C00743=24023,61091,-95954,71320,-125497,-86258,0
C00744=47988,53738,-118403,64043,-120090,-93197,0
C00745=47969,53677,-118607,64035,-120007,-93252,0
C00746=24001,61005,-96191,71299,-125419,-86322,0
C00747=23979,60920,-96427,71278,-125340,-86384,0
C00748=47959,53616,-118810,64017,-119928,-93309,0
C00749=47965,53556,-119011,63982,-119855,-93367,0
C00750=23938,60841,-96646,71279,-125255,-86439,0
C00751=23896,60763,-96863,71283,-125169,-86492,0
C00752=47974,53496,-119211,63945,-119783,-93425,0
C00753=48004,53437,-119411,63884,-119719,-93487,0
C00754=23849,60687,-97075,71292,-125082,-86544,0
C00755=23834,60662,-97143,71295,-125055,-86561,0
C00756=23790,60615,-97275,71316,-124991,-86591,0
C00757=48035,53378,-119610,63823,-119656,-93548,0
C00758=48091,53320,-119808,63734,-119602,-93612,0
C00759=23724,60545,-97468,71348,-124899,-86634,0
C00760=23711,60532,-97506,71354,-124881,-86643,0
C00761=23641,60482,-97645,71401,-124802,-86670,0
C00762=48149,53263,-120004,63643,-119548,-93677,0
C00763=48238,53206,-120198,63519,-119506,-93744,0
C00764=23551,60420,-97816,71461,-124702,-86703,0
C00765=23436,60368,-97962,71552,-124595,-86725,0
C00766=48338,53150,-120391,63384,-119469,-93813,0
C00767=48473,53095,-120582,63209,-119443,-93887,0
C00768=23301,60322,-98088,71667,-124481,-86739,0
C00769=23194,60294,-98165,71761,-124398,-86743,0
C00770=23131,60288,-98180,71823,-124357,-86737,0
C00771=48657,53042,-120768,62982,-119437,-93964,0
C00772=48736,53022,-120839,62886,-119437,-93996,0
C00773=48942,52993,-120945,62645,-119469,-94054,0
C00774=22868,60287,-98181,72089,-124204,-86695,0
C00775=22798,60292,-98165,72162,-124169,-86679,0
C00776=22666,60326,-98070,72312,-124118,-86631,0
C00777=22702,60253,-98275,72240,-124082,-86695,0
C00778=49183,52943,-121124,62357,-119483,-94138,0
C00779=49183,52942,-121127,62356,-119482,-94138,0
C00780=49239,52943,-121127,62294,-119502,-94147,0
C00781=49127,52884,-121328,62390,-119383,-94188,0
C00782=22756,60143,-98582,72132,-124030,-86790,0
C00783=22810,60035,-98889,72024,-123977,-86886,0
C00784=49009,52823,-121536,62492,-119261,-94231,0
C00785=48890,52762,-121744,62594,-119139,-94275,0
C00786=22865,59926,-99195,71916,-123923,-86981,0
C00787=22920,59818,-99500,71808,-123870,-87077,0
C00788=48771,52701,-121951,62697,-119016,-94318,0
C00789=48652,52641,-122158,62801,-118894,-94362,0
C00790=22975,59711,-99804,71700,-123816,-87172,0
C00791=23030,59604,-100107,71592,-123762,-87266,0
C00792=48532,52581,-122363,62906,-118772,-94405,0
C00793=48411,52521,-122569,63012,-118650,-94449,0
C00794=23086,59498,-100409,71484,-123709,-87361,0
C00795=23142,59393,-100710,71375,-123655,-87455,0
C00796=48290,52462,-122773,63118,-118530,-94492,0
C00797=48168,52404,-122977,63225,-118409,-94536,0
C00798=23198,59287,-101011,71267,-123601,-87549,0
C00799=23255,59182,-101310,71158,-123546,-87643,0
C00800=48046,52345,-123180,63334,-118288,-94579,0
C00801=47923,52287,-123383,63442,-118168,-94622,0
C00802=23311,59078,-101609,71050,-123492,-87737,0
C00803=23368,58975,-101907,70941,-123438,-87831,0
C00804=47800,52230,-123585,63552,-118048,-94666,0
C00805=47676,52172,-123786,63663,-117929,-94709,0
C00806=23425,58871,-102204,70833,-123383,-87924,0
C00807=23483,58769,-102500,70724,-123329,-88017,0
C00808=47551,52115,-123986,63774,-117809,-94753,0
C00809=47426,52059,-124186,63887,-117690,-94796,0
C00810=23541,58666,-102796,70615,-123273,-88110,0
C00811=23598,58565,-103090,70506,-123218,-88203,0
C00812=47301,52003,-124386,64000,-117571,-94839,0
C00813=47175,51947,-124585,64114,-117453,-94883,0
C00814=23657,58463,-103384,70397,-123163,-88296,0
C00815=23715,58362,-103677,70288,-123108,-88388,0
C00816=47048,51891,-124782,64229,-117336,-94926,0
C00817=46921,51836,-124980,64344,-117217,-94969,0
C00818=23774,58262,-103969,70179,-123053,-88480,0
C00819=23833,58162,-104260,70069,-122996,-88572,0
C00820=46793,51781,-125176,64461,-117100,-95013,0
C00821=46664,51727,-125372,64578,-116983,-95056,0
C00822=23893,58063,-104551,69960,-122941,-88664,0
C00823=23952,57964,-104840,69850,-122885,-88755,0
C00824=46535,51673,-125567,64697,-116867,-95099,0
C00825=46406,51619,-125762,64816,-116751,-95143,0
C00826=24012,57866,-105129,69741,-122829,-88846,0
C00827=24073,57768,-105417,69631,-122772,-88938,0
C00828=46276,51566,-125955,64936,-116635,-95186,0
C00829=46145,51513,-126150,65057,-116519,-95229,0
C00830=24133,57670,-105705,69521,-122716,-89029,0
C00831=24194,57573,-105991,69411,-122660,-89120,0
C00832=38915,55283,-113204,52158,-126367,-93683,0
C00833=38787,55224,-113386,52273,-126238,-93702,0
C00834=24255,57477,-106277,69301,-122603,-89210,0
C00835=24316,57380,-106562,69191,-122546,-89301,0
C00836=38658,55165,-113568,52388,-126109,-93722,0
C00837=38530,55107,-113749,52503,-125981,-93741,0
C00838=24378,57285,-106847,69080,-122490,-89391,0
C00839=24440,57190,-107130,68970,-122432,-89481,0
C00840=38400,55049,-113929,52619,-125853,-93761,0
C00841=38271,54991,-114109,52736,-125726,-93780,0
C00842=24502,57095,-107413,68859,-122375,-89571,0
C00843=24565,57001,-107695,68748,-122317,-89661,0
C00844=38140,54934,-114287,52854,-125599,-93800,0
C00845=38010,54877,-114465,52972,-125472,-93819,0
C00846=24628,56907,-107976,68638,-122260,-89750,0
C00847=24691,56813,-108257,68527,-122201,-89840,0
C00848=37879,54820,-114643,53091,-125345,-93838,0
C00849=37747,54764,-114819,53210,-125219,-93858,0
C00850=24754,56721,-108537,68415,-122144,-89929,0
C00851=24818,56628,-108816,68304,-122085,-90019,0
C00852=37616,54708,-114995,53330,-125094,-93877,0
C00853=37483,54652,-115170,53451,-124968,-93896,0
C00854=24882,56536,-109095,68192,-122028,-90107,0
C00855=24947,56445,-109372,68081,-121969,-90196,0
C00856=37350,54597,-115344,53572,-124843,-93915,0
C00857=37217,54542,-115518,53694,-124718,-93934,0
C00858=25011,56354,-109650,67969,-121910,-90285,0
C00859=25076,56263,-109926,67857,-121851,-90373,0
C00860=37083,54487,-115691,53817,-124594,-93953,0
C00861=36949,54433,-115862,53940,-124470,-93972,0
C00862=25142,56173,-110201,67745,-121792,-90461,0
C00863=25207,56083,-110476,67633,-121732,-90549,0
C00864=36815,54378,-116034,54064,-124346,-93992,0
C00865=36680,54325,-116205,54188,-124221,-94011,0
C00866=25273,55994,-110751,67520,-121674,-90637,0
C00867=25340,55905,-111024,67407,-121614,-90725,0
C00868=36544,54271,-116375,54314,-124098,-94029,0
C00869=36408,54218,-116544,54440,-123975,-94048,0
C00870=25406,55816,-111297,67294,-121554,-90813,0
C00871=25473,55729,-111569,67181,-121494,-90900,0
C00872=36272,54166,-116712,54566,-123854,-94068,0
C00873=36135,54113,-116879,54693,-123731,-94086,0
C00874=25541,55641,-111841,67068,-121434,-90988,0
C00875=25608,55554,-112112,66955,-121374,-91075,0
C00876=35998,54061,-117047,54821,-123609,-94105,0
C00877=35860,54010,-117213,54950,-123487,-94124,0
C00878=25676,55467,-112382,66841,-121313,-91162,0
C00879=25745,55381,-112651,66727,-121252,-91249,0
C00880=35722,53958,-117378,55079,-123366,-94143,0
C00881=35583,53907,-117543,55209,-123245,-94162,0
C00882=25813,55295,-112920,66613,-121191,-91335,0
C00883=25882,55210,-113188,66499,-121130,-91422,0
C00884=35444,53856,-117707,55339,-123124,-94181,0
C00885=35305,53806,-117870,55470,-123004,-94199,0
C00886=25952,55125,-113456,66385,-121069,-91508,0
C00887=26021,55041,-113723,66270,-121007,-91595,0
C00888=35165,53756,-118033,55602,-122884,-94218,0
C00889=35024,53706,-118194,55734,-122764,-94236,0
C00890=26091,54957,-113989,66155,-120945,-91680,0
C00891=26162,54873,-114255,66040,-120884,-91766,0
C00892=34883,53657,-118355,55867,-122646,-94256,0
C00893=34742,53607,-118516,56001,-122526,-94274,0
C00894=26233,54790,-114519,65925,-120821,-91852,0
C00895=26304,54707,-114784,65810,-120759,-91937,0
C00896=34600,53559,-118676,56136,-122408,-94293,0
C00897=34458,53510,-118834,56271,-122290,-94311,0
C00898=26375,54625,-115048,65694,-120697,-92023,0
C00899=26447,54543,-115311,65578,-120634,-92109,0
C00900=34315,53462,-118992,56406,-122171,-94330,0
C00901=34172,53414,-119149,56543,-122054,-94348,0
C00902=26519,54462,-115573,65462,-120571,-92194,0
C00903=26592,54381,-115835,65346,-120507,-92279,0
C00904=34028,53366,-119305,56680,-121937,-94367,0
C00905=33884,53319,-119462,56817,-121820,-94385,0
C00906=26665,54300,-116096,65229,-120444,-92363,0
C00907=26738,54220,-116357,65112,-120381,-92449,0
C00908=33739,53272,-119617,56956,-121704,-94404,0
C00909=33594,53226,-119771,57095,-121588,-94422,0
C00910=26812,54140,-116616,64995,-120317,-92533,0
C00911=26886,54061,-116875,64878,-120253,-92618,0
C00912=33449,53179,-119924,57234,-121471,-94441,0
C00913=33302,53134,-120076,57374,-121357,-94459,0
C00914=26960,53982,-117133,64760,-120189,-92702,0
C00915=27035,53904,-117392,64642,-120125,-92786,0
C00916=33156,53088,-120229,57515,-121241,-94477,0
C00917=33009,53042,-120380,57657,-121126,-94495,0
C00918=27110,53826,-117649,64524,-120059,-92870,0
C00919=27186,53748,-117906,64406,-119995,-92954,0
C00920=32862,52997,-120530,57799,-121012,-94514,0
C00921=32714,52953,-120681,57942,-120898,-94532,0
C00922=27262,53671,-118162,64287,-119929,-93038,0
C00923=27338,53594,-118418,64168,-119864,-93121,0
C00924=32565,52908,-120829,58086,-120784,-94550,0
C00925=32417,52864,-120979,58230,-120671,-94568,0
C00926=27415,53518,-118673,64049,-119798,-93205,0
C00927=27492,53442,-118927,63930,-119733,-93288,0
C00928=29484,53152,-119939,61610,-120078,-93854,0
C00929=29348,53143,-119967,61755,-120017,-93843,0
C00930=29237,53124,-120029,61868,-119952,-93845,0
C00931=27570,53367,-119181,63810,-119666,-93371,0
C00932=27648,53292,-119434,63690,-119600,-93454,0
C00933=29053,53088,-120149,62054,-119839,-93852,0
C00934=28906,53047,-120287,62196,-119733,-93871,0
C00935=27726,53217,-119687,63570,-119533,-93537,0
C00936=27805,53143,-119939,63449,-119466,-93620,0
C00937=28788,53002,-120437,62305,-119631,-93897,0
C00938=28679,52956,-120591,62404,-119531,-93925,0
C00939=27884,53069,-120190,63328,-119400,-93703,0
C00940=27964,52996,-120441,63207,-119332,-93785,0
C00941=28598,52906,-120760,62469,-119436,-93963,0
C00942=28519,52856,-120929,62533,-119342,-94000,0
C00943=28044,52923,-120691,63086,-119265,-93867,0
C00944=28124,52851,-120941,62964,-119197,-93950,0
C00945=28463,52803,-121111,62570,-119251,-94044,0
C00946=28431,52773,-121215,62591,-119198,-94069,0
C00947=28356,52785,-121170,62680,-119190,-94046,0
C00948=28336,52761,-121255,62690,-119149,-94068,0
C00949=28206,52779,-121190,62842,-119128,-94032,0
C00950=30856,52503,-122197,59790,-119634,-94679,0
C00951=31056,52481,-122279,59558,-119665,-94730,0
C00952=31209,52522,-122137,59408,-119775,-94712,0
C00953=30866,52561,-121997,59806,-119720,-94625,0
C00954=30874,52612,-121820,59821,-119797,-94577,0
C00955=30870,52619,-121793,59829,-119806,-94569,0
C00956=31362,52564,-121996,59258,-119887,-94694,0
C00957=31514,52606,-121852,59109,-119997,-94676,0
C00958=30838,52682,-121575,59894,-119886,-94503,0
C00959=30806,52745,-121357,59960,-119966,-94438,0
C00960=31665,52648,-121708,58961,-120109,-94658,0
C00961=31817,52691,-121563,58813,-120220,-94640,0
C00962=30743,52812,-121124,60061,-120040,-94365,0
C00963=30686,52870,-120924,60151,-120103,-94301,0
C00964=30670,52880,-120888,60174,-120112,-94288,0
C00965=31967,52734,-121419,58667,-120333,-94622,0
C00966=32117,52777,-121273,58520,-120444,-94604,0
C00967=30557,52954,-120633,60334,-120178,-94201,0
C00968=30523,52976,-120557,60381,-120197,-94175,0
C00969=30389,53035,-120352,60558,-120234,-94099,0
C00970=32267,52820,-121126,58375,-120557,-94586,0
C00971=32417,52864,-120979,58230,-120671,-94568,0
C00972=28376,52719,-121400,62627,-119107,-94115,0
C00973=28356,52694,-121485,62637,-119066,-94137,0
C00974=28336,52669,-121570,62648,-119026,-94158,0
C00975=28337,52667,-121580,62646,-119023,-94160,0
C00976=28343,52645,-121655,62630,-118995,-94183,0
C00977=28428,52534,-122041,62484,-118872,-94305,0
C00978=28425,52521,-122090,62481,-118853,-94318,0
C00979=28416,52479,-122232,62473,-118793,-94358,0
C00980=28426,52464,-122285,62455,-118776,-94375,0
//INST
///DATE 2025/02/20 16:20
///COMM Generated using RoboDK
///ATTR SC,RW
///GROUP1 RB1
NOP
'Program generated by RoboDK v
'5.9.0 for Yaskawa SIA10D on 2
'0/02/2025 16:20:52
'Using nominal kinematics.
CALL JOB:ONSTART
CALL JOB:MCODEHA
CALL JOB:SETRPM(
CALL JOB:MCODEHA
'Using Printing Frame (targets
' wrt base):
'471.7,0.0,-333.4,0.0,0.6,180.
'0
'Tool MDPH2 should be close to
':
'-226.5,0.0,70.1,0.0,-90.0,0.0
'Show MDPH2
MOVJ C00000 VJ=50.00 PL=1
MOVL C00001 V=80.0 PL=1
CALL JOB:SETRPM(
CALL JOB:MCODEHA
CALL JOB:MCODEHA
CALL JOB:EXTRUDE
MOVL C00002 V=130.0 PL=1
CALL JOB:EXTRUDE
CALL JOB:EXTRUDE
CALL JOB:EXTRUDE
CALL JOB:EXTRUDE
MOVL C00003 V=30.0 PL=1
CALL JOB:EXTRUDE
MOVL C00004 V=30.0 PL=1
CALL JOB:EXTRUDE
MOVL C00005 V=30.0 PL=1
CALL JOB:EXTRUDE
MOVL C00006 V=30.0 PL=1
CALL JOB:EXTRUDE
MOVL C00007 V=30.0 PL=1
CALL JOB:EXTRUDE
MOVL C00008 V=30.0 PL=1
CALL JOB:EXTRUDE
MOVL C00009 V=30.0 PL=1
CALL JOB:EXTRUDE
MOVL C00010 V=30.0 PL=1
CALL JOB:EXTRUDE
MOVL C00011 V=30.0 PL=1
CALL JOB:EXTRUDE
MOVL C00012 V=30.0 PL=1
CALL JOB:EXTRUDE
MOVL C00013 V=30.0 PL=1
CALL JOB:EXTRUDE
MOVL C00014 V=30.0 PL=1
CALL JOB:EXTRUDE
MOVL C00015 V=30.0 PL=1
CALL JOB:EXTRUDE
MOVL C00016 V=30.0 PL=1
CALL JOB:EXTRUDE
MOVL C00017 V=30.0 PL=1
CALL JOB:EXTRUDE
MOVL C00018 V=30.0 PL=1
CALL JOB:EXTRUDE
MOVL C00019 V=30.0 PL=1
CALL JOB:EXTRUDE
MOVL C00020 V=30.0 PL=1
CALL JOB:EXTRUDE
MOVL C00021 V=30.0 PL=1
CALL JOB:EXTRUDE
MOVL C00022 V=30.0 PL=1
CALL JOB:EXTRUDE
MOVL C00023 V=30.0 PL=1
CALL JOB:EXTRUDE
MOVL C00024 V=30.0 PL=1
CALL JOB:EXTRUDE
MOVL C00025 V=30.0 PL=1
CALL JOB:EXTRUDE
MOVL C00026 V=30.0 PL=1
CALL JOB:EXTRUDE
CALL JOB:EXTRUDE
MOVL C00027 V=130.0 PL=1
CALL JOB:EXTRUDE
CALL JOB:EXTRUDE
MOVL C00028 V=30.0 PL=1
CALL JOB:EXTRUDE
MOVL C00029 V=30.0 PL=1
CALL JOB:EXTRUDE
MOVL C00030 V=30.0 PL=1
CALL JOB:EXTRUDE
MOVL C00031 V=30.0 PL=1
CALL JOB:EXTRUDE
MOVL C00032 V=30.0 PL=1
CALL JOB:EXTRUDE
MOVL C00033 V=30.0 PL=1
CALL JOB:EXTRUDE
MOVL C00034 V=30.0 PL=1
CALL JOB:EXTRUDE
MOVL C00035 V=30.0 PL=1
CALL JOB:EXTRUDE
MOVL C00036 V=30.0 PL=1
CALL JOB:EXTRUDE
MOVL C00037 V=30.0 PL=1
CALL JOB:EXTRUDE
MOVL C00038 V=30.0 PL=1
CALL JOB:EXTRUDE
MOVL C00039 V=30.0 PL=1
CALL JOB:EXTRUDE
MOVL C00040 V=30.0 PL=1
CALL JOB:EXTRUDE
MOVL C00041 V=30.0 PL=1
CALL JOB:EXTRUDE
MOVL C00042 V=30.0 PL=1
CALL JOB:EXTRUDE
MOVL C00043 V=30.0 PL=1
CALL JOB:EXTRUDE
MOVL C00044 V=30.0 PL=1
CALL JOB:EXTRUDE
MOVL C00045 V=30.0 PL=1
CALL JOB:EXTRUDE
MOVL C00046 V=30.0 PL=1
CALL JOB:EXTRUDE
MOVL C00047 V=30.0 PL=1
CALL JOB:EXTRUDE
MOVL C00048 V=30.0 PL=1
CALL JOB:EXTRUDE
MOVL C00049 V=30.0 PL=1
CALL JOB:EXTRUDE
MOVL C00050 V=30.0 PL=1
CALL JOB:EXTRUDE
MOVL C00051 V=30.0 PL=1
CALL JOB:EXTRUDE
MOVL C00052 V=30.0 PL=1
CALL JOB:EXTRUDE
MOVL C00053 V=30.0 PL=1
CALL JOB:EXTRUDE
MOVL C00054 V=30.0 PL=1
CALL JOB:EXTRUDE
MOVL C00055 V=30.0 PL=1
CALL JOB:EXTRUDE
MOVL C00056 V=30.0 PL=1
CALL JOB:EXTRUDE
MOVL C00057 V=30.0 PL=1
CALL JOB:EXTRUDE
MOVL C00058 V=30.0 PL=1
CALL JOB:EXTRUDE
MOVL C00059 V=30.0 PL=1
MOVL C00060 V=130.0 PL=1
CALL JOB:EXTRUDE
MOVL C00061 V=30.0 PL=1
CALL JOB:EXTRUDE
MOVL C00062 V=30.0 PL=1
CALL JOB:EXTRUDE
MOVL C00063 V=30.0 PL=1
CALL JOB:EXTRUDE
MOVL C00064 V=30.0 PL=1
CALL JOB:EXTRUDE
MOVL C00065 V=30.0 PL=1
CALL JOB:EXTRUDE
MOVL C00066 V=30.0 PL=1
CALL JOB:EXTRUDE
MOVL C00067 V=30.0 PL=1
CALL JOB:EXTRUDE
MOVL C00068 V=30.0 PL=1
CALL JOB:EXTRUDE
MOVL C00069 V=30.0 PL=1
CALL JOB:EXTRUDE
MOVL C00070 V=30.0 PL=1
CALL JOB:EXTRUDE
MOVL C00071 V=30.0 PL=1
CALL JOB:EXTRUDE
MOVL C00072 V=30.0 PL=1
CALL JOB:EXTRUDE
MOVL C00073 V=30.0 PL=1
CALL JOB:EXTRUDE
MOVL C00074 V=30.0 PL=1
CALL JOB:EXTRUDE
MOVL C00075 V=30.0 PL=1
CALL JOB:EXTRUDE
MOVL C00076 V=30.0 PL=1
CALL JOB:EXTRUDE
MOVL C00077 V=30.0 PL=1
CALL JOB:EXTRUDE
MOVL C00078 V=30.0 PL=1
CALL JOB:EXTRUDE
MOVL C00079 V=30.0 PL=1
CALL JOB:EXTRUDE
MOVL C00080 V=30.0 PL=1
CALL JOB:EXTRUDE
MOVL C00081 V=30.0 PL=1
CALL JOB:EXTRUDE
MOVL C00082 V=30.0 PL=1
CALL JOB:EXTRUDE
MOVL C00083 V=30.0 PL=1
CALL JOB:EXTRUDE
MOVL C00084 V=30.0 PL=1
CALL JOB:EXTRUDE
MOVL C00085 V=30.0 PL=1
CALL JOB:EXTRUDE
MOVL C00086 V=30.0 PL=1
CALL JOB:EXTRUDE
MOVL C00087 V=30.0 PL=1
CALL JOB:EXTRUDE
MOVL C00088 V=30.0 PL=1
CALL JOB:EXTRUDE
MOVL C00089 V=30.0 PL=1
CALL JOB:EXTRUDE
MOVL C00090 V=30.0 PL=1
CALL JOB:EXTRUDE
MOVL C00091 V=30.0 PL=1
CALL JOB:EXTRUDE
MOVL C00092 V=30.0 PL=1
MOVL C00093 V=130.0 PL=1
CALL JOB:EXTRUDE
CALL JOB:EXTRUDE
MOVL C00094 V=130.0 PL=1
CALL JOB:EXTRUDE
CALL JOB:EXTRUDE
MOVL C00095 V=30.0 PL=1
CALL JOB:EXTRUDE
MOVL C00096 V=30.0 PL=1
CALL JOB:EXTRUDE
MOVL C00097 V=30.0 PL=1
CALL JOB:EXTRUDE
MOVL C00098 V=30.0 PL=1
CALL JOB:EXTRUDE
MOVL C00099 V=30.0 PL=1
CALL JOB:EXTRUDE
MOVL C00100 V=30.0 PL=1
CALL JOB:EXTRUDE
MOVL C00101 V=30.0 PL=1
CALL JOB:EXTRUDE
MOVL C00102 V=30.0 PL=1
CALL JOB:EXTRUDE
CALL JOB:EXTRUDE
MOVL C00103 V=130.0 PL=1
CALL JOB:EXTRUDE
CALL JOB:EXTRUDE
MOVL C00104 V=30.0 PL=1
CALL JOB:EXTRUDE
MOVL C00105 V=30.0 PL=1
CALL JOB:EXTRUDE
MOVL C00106 V=30.0 PL=1
CALL JOB:EXTRUDE
MOVL C00107 V=30.0 PL=1
CALL JOB:EXTRUDE
MOVL C00108 V=30.0 PL=1
CALL JOB:EXTRUDE
MOVL C00109 V=30.0 PL=1
CALL JOB:EXTRUDE
MOVL C00110 V=30.0 PL=1
CALL JOB:EXTRUDE
MOVL C00111 V=30.0 PL=1
CALL JOB:EXTRUDE
MOVL C00112 V=30.0 PL=1
CALL JOB:EXTRUDE
MOVL C00113 V=30.0 PL=1
CALL JOB:EXTRUDE
MOVL C00114 V=30.0 PL=1
CALL JOB:EXTRUDE
MOVL C00115 V=30.0 PL=1
CALL JOB:EXTRUDE
MOVL C00116 V=30.0 PL=1
CALL JOB:EXTRUDE
MOVL C00117 V=30.0 PL=1
CALL JOB:EXTRUDE
MOVL C00118 V=30.0 PL=1
CALL JOB:EXTRUDE
MOVL C00119 V=30.0 PL=1
CALL JOB:EXTRUDE
MOVL C00120 V=30.0 PL=1
CALL JOB:EXTRUDE
MOVL C00121 V=30.0 PL=1
CALL JOB:EXTRUDE
MOVL C00122 V=30.0 PL=1
CALL JOB:EXTRUDE
MOVL C00123 V=30.0 PL=1
CALL JOB:EXTRUDE
MOVL C00124 V=30.0 PL=1
CALL JOB:EXTRUDE
MOVL C00125 V=30.0 PL=1
CALL JOB:EXTRUDE
MOVL C00126 V=30.0 PL=1
CALL JOB:EXTRUDE
MOVL C00127 V=30.0 PL=1
CALL JOB:EXTRUDE
MOVL C00128 V=30.0 PL=1
CALL JOB:EXTRUDE
MOVL C00129 V=30.0 PL=1
CALL JOB:EXTRUDE
MOVL C00130 V=30.0 PL=1
CALL JOB:EXTRUDE
MOVL C00131 V=30.0 PL=1
CALL JOB:EXTRUDE
MOVL C00132 V=30.0 PL=1
CALL JOB:EXTRUDE
MOVL C00133 V=30.0 PL=1
CALL JOB:EXTRUDE
MOVL C00134 V=30.0 PL=1
CALL JOB:EXTRUDE
MOVL C00135 V=30.0 PL=1
MOVL C00136 V=130.0 PL=1
CALL JOB:EXTRUDE
MOVL C00137 V=30.0 PL=1
CALL JOB:EXTRUDE
MOVL C00138 V=30.0 PL=1
CALL JOB:EXTRUDE
MOVL C00139 V=30.0 PL=1
CALL JOB:EXTRUDE
MOVL C00140 V=30.0 PL=1
CALL JOB:EXTRUDE
MOVL C00141 V=30.0 PL=1
CALL JOB:EXTRUDE
MOVL C00142 V=30.0 PL=1
CALL JOB:EXTRUDE
MOVL C00143 V=30.0 PL=1
CALL JOB:EXTRUDE
MOVL C00144 V=30.0 PL=1
CALL JOB:EXTRUDE
MOVL C00145 V=30.0 PL=1
CALL JOB:EXTRUDE
MOVL C00146 V=30.0 PL=1
CALL JOB:EXTRUDE
MOVL C00147 V=30.0 PL=1
CALL JOB:EXTRUDE
MOVL C00148 V=30.0 PL=1
CALL JOB:EXTRUDE
MOVL C00149 V=30.0 PL=1
CALL JOB:EXTRUDE
MOVL C00150 V=30.0 PL=1
CALL JOB:EXTRUDE
MOVL C00151 V=30.0 PL=1
CALL JOB:EXTRUDE
MOVL C00152 V=30.0 PL=1
CALL JOB:EXTRUDE
MOVL C00153 V=30.0 PL=1
CALL JOB:EXTRUDE
MOVL C00154 V=30.0 PL=1
CALL JOB:EXTRUDE
MOVL C00155 V=30.0 PL=1
CALL JOB:EXTRUDE
MOVL C00156 V=30.0 PL=1
CALL JOB:EXTRUDE
MOVL C00157 V=30.0 PL=1
CALL JOB:EXTRUDE
MOVL C00158 V=30.0 PL=1
CALL JOB:EXTRUDE
MOVL C00159 V=30.0 PL=1
CALL JOB:EXTRUDE
MOVL C00160 V=30.0 PL=1
CALL JOB:EXTRUDE
MOVL C00161 V=30.0 PL=1
CALL JOB:EXTRUDE
MOVL C00162 V=30.0 PL=1
CALL JOB:EXTRUDE
MOVL C00163 V=30.0 PL=1
CALL JOB:EXTRUDE
MOVL C00164 V=30.0 PL=1
CALL JOB:EXTRUDE
MOVL C00165 V=30.0 PL=1
CALL JOB:EXTRUDE
MOVL C00166 V=30.0 PL=1
CALL JOB:EXTRUDE
MOVL C00167 V=30.0 PL=1
CALL JOB:EXTRUDE
MOVL C00168 V=30.0 PL=1
MOVL C00169 V=130.0 PL=1
CALL JOB:EXTRUDE
CALL JOB:EXTRUDE
MOVL C00170 V=130.0 PL=1
CALL JOB:EXTRUDE
CALL JOB:EXTRUDE
MOVL C00171 V=30.0 PL=1
CALL JOB:EXTRUDE
MOVL C00172 V=30.0 PL=1
CALL JOB:EXTRUDE
MOVL C00173 V=30.0 PL=1
CALL JOB:EXTRUDE
MOVL C00174 V=30.0 PL=1
CALL JOB:EXTRUDE
MOVL C00175 V=30.0 PL=1
CALL JOB:EXTRUDE
MOVL C00176 V=30.0 PL=1
CALL JOB:EXTRUDE
MOVL C00177 V=30.0 PL=1
CALL JOB:EXTRUDE
MOVL C00178 V=30.0 PL=1
CALL JOB:EXTRUDE
MOVL C00179 V=30.0 PL=1
CALL JOB:EXTRUDE
MOVL C00180 V=30.0 PL=1
CALL JOB:EXTRUDE
MOVL C00181 V=30.0 PL=1
CALL JOB:EXTRUDE
MOVL C00182 V=30.0 PL=1
CALL JOB:EXTRUDE
MOVL C00183 V=30.0 PL=1
CALL JOB:EXTRUDE
MOVL C00184 V=30.0 PL=1
CALL JOB:EXTRUDE
MOVL C00185 V=30.0 PL=1
CALL JOB:EXTRUDE
MOVL C00186 V=30.0 PL=1
CALL JOB:EXTRUDE
MOVL C00187 V=30.0 PL=1
CALL JOB:EXTRUDE
MOVL C00188 V=30.0 PL=1
CALL JOB:EXTRUDE
MOVL C00189 V=30.0 PL=1
CALL JOB:EXTRUDE
MOVL C00190 V=30.0 PL=1
CALL JOB:EXTRUDE
MOVL C00191 V=30.0 PL=1
CALL JOB:EXTRUDE
MOVL C00192 V=30.0 PL=1
CALL JOB:EXTRUDE
MOVL C00193 V=30.0 PL=1
CALL JOB:EXTRUDE
MOVL C00194 V=30.0 PL=1
CALL JOB:EXTRUDE
MOVL C00195 V=30.0 PL=1
CALL JOB:EXTRUDE
MOVL C00196 V=30.0 PL=1
CALL JOB:EXTRUDE
MOVL C00197 V=30.0 PL=1
CALL JOB:EXTRUDE
MOVL C00198 V=30.0 PL=1
CALL JOB:EXTRUDE
MOVL C00199 V=30.0 PL=1
CALL JOB:EXTRUDE
MOVL C00200 V=30.0 PL=1
CALL JOB:EXTRUDE
MOVL C00201 V=30.0 PL=1
CALL JOB:EXTRUDE
MOVL C00202 V=30.0 PL=1
MOVL C00203 V=130.0 PL=1
CALL JOB:EXTRUDE
MOVL C00204 V=30.0 PL=1
CALL JOB:EXTRUDE
MOVL C00205 V=30.0 PL=1
CALL JOB:EXTRUDE
MOVL C00206 V=30.0 PL=1
CALL JOB:EXTRUDE
MOVL C00207 V=30.0 PL=1
CALL JOB:EXTRUDE
MOVL C00208 V=30.0 PL=1
CALL JOB:EXTRUDE
MOVL C00209 V=30.0 PL=1
CALL JOB:EXTRUDE
MOVL C00210 V=30.0 PL=1
CALL JOB:EXTRUDE
MOVL C00211 V=30.0 PL=1
CALL JOB:EXTRUDE
MOVL C00212 V=30.0 PL=1
CALL JOB:EXTRUDE
MOVL C00213 V=30.0 PL=1
CALL JOB:EXTRUDE
MOVL C00214 V=30.0 PL=1
CALL JOB:EXTRUDE
MOVL C00215 V=30.0 PL=1
CALL JOB:EXTRUDE
MOVL C00216 V=30.0 PL=1
CALL JOB:EXTRUDE
MOVL C00217 V=30.0 PL=1
CALL JOB:EXTRUDE
MOVL C00218 V=30.0 PL=1
CALL JOB:EXTRUDE
MOVL C00219 V=30.0 PL=1
CALL JOB:EXTRUDE
MOVL C00220 V=30.0 PL=1
CALL JOB:EXTRUDE
MOVL C00221 V=30.0 PL=1
CALL JOB:EXTRUDE
MOVL C00222 V=30.0 PL=1
CALL JOB:EXTRUDE
MOVL C00223 V=30.0 PL=1
CALL JOB:EXTRUDE
MOVL C00224 V=30.0 PL=1
CALL JOB:EXTRUDE
MOVL C00225 V=30.0 PL=1
CALL JOB:EXTRUDE
MOVL C00226 V=30.0 PL=1
CALL JOB:EXTRUDE
MOVL C00227 V=30.0 PL=1
CALL JOB:EXTRUDE
MOVL C00228 V=30.0 PL=1
CALL JOB:EXTRUDE
MOVL C00229 V=30.0 PL=1
CALL JOB:EXTRUDE
MOVL C00230 V=30.0 PL=1
CALL JOB:EXTRUDE
MOVL C00231 V=30.0 PL=1
CALL JOB:EXTRUDE
MOVL C00232 V=30.0 PL=1
CALL JOB:EXTRUDE
MOVL C00233 V=30.0 PL=1
CALL JOB:EXTRUDE
MOVL C00234 V=30.0 PL=1
CALL JOB:EXTRUDE
MOVL C00235 V=30.0 PL=1
MOVL C00236 V=130.0 PL=1
CALL JOB:EXTRUDE
CALL JOB:EXTRUDE
MOVL C00237 V=130.0 PL=1
CALL JOB:EXTRUDE
CALL JOB:EXTRUDE
MOVL C00238 V=30.0 PL=1
CALL JOB:EXTRUDE
MOVL C00239 V=30.0 PL=1
CALL JOB:EXTRUDE
MOVL C00240 V=30.0 PL=1
CALL JOB:EXTRUDE
MOVL C00241 V=30.0 PL=1
CALL JOB:EXTRUDE
MOVL C00242 V=30.0 PL=1
CALL JOB:EXTRUDE
MOVL C00243 V=30.0 PL=1
CALL JOB:EXTRUDE
MOVL C00244 V=30.0 PL=1
CALL JOB:EXTRUDE
MOVL C00245 V=30.0 PL=1
CALL JOB:EXTRUDE
MOVL C00246 V=30.0 PL=1
CALL JOB:EXTRUDE
MOVL C00247 V=30.0 PL=1
CALL JOB:EXTRUDE
MOVL C00248 V=30.0 PL=1
CALL JOB:EXTRUDE
MOVL C00249 V=30.0 PL=1
CALL JOB:EXTRUDE
MOVL C00250 V=30.0 PL=1
CALL JOB:EXTRUDE
MOVL C00251 V=30.0 PL=1
CALL JOB:EXTRUDE
MOVL C00252 V=30.0 PL=1
CALL JOB:EXTRUDE
MOVL C00253 V=30.0 PL=1
CALL JOB:EXTRUDE
MOVL C00254 V=30.0 PL=1
CALL JOB:EXTRUDE
MOVL C00255 V=30.0 PL=1
CALL JOB:EXTRUDE
MOVL C00256 V=30.0 PL=1
CALL JOB:EXTRUDE
MOVL C00257 V=30.0 PL=1
CALL JOB:EXTRUDE
MOVL C00258 V=30.0 PL=1
CALL JOB:EXTRUDE
MOVL C00259 V=30.0 PL=1
CALL JOB:EXTRUDE
MOVL C00260 V=30.0 PL=1
CALL JOB:EXTRUDE
MOVL C00261 V=30.0 PL=1
CALL JOB:EXTRUDE
MOVL C00262 V=30.0 PL=1
CALL JOB:EXTRUDE
MOVL C00263 V=30.0 PL=1
CALL JOB:EXTRUDE
MOVL C00264 V=30.0 PL=1
CALL JOB:EXTRUDE
MOVL C00265 V=30.0 PL=1
CALL JOB:EXTRUDE
MOVL C00266 V=30.0 PL=1
CALL JOB:EXTRUDE
MOVL C00267 V=30.0 PL=1
CALL JOB:EXTRUDE
MOVL C00268 V=30.0 PL=1
CALL JOB:EXTRUDE
MOVL C00269 V=30.0 PL=1
CALL JOB:EXTRUDE
MOVL C00270 V=30.0 PL=1
CALL JOB:EXTRUDE
MOVL C00271 V=30.0 PL=1
CALL JOB:EXTRUDE
MOVL C00272 V=30.0 PL=1
CALL JOB:EXTRUDE
MOVL C00273 V=30.0 PL=1
CALL JOB:EXTRUDE
MOVL C00274 V=30.0 PL=1
CALL JOB:EXTRUDE
MOVL C00275 V=30.0 PL=1
CALL JOB:EXTRUDE
MOVL C00276 V=30.0 PL=1
CALL JOB:EXTRUDE
MOVL C00277 V=30.0 PL=1
CALL JOB:EXTRUDE
MOVL C00278 V=30.0 PL=1
CALL JOB:EXTRUDE
MOVL C00279 V=30.0 PL=1
CALL JOB:EXTRUDE
MOVL C00280 V=30.0 PL=1
CALL JOB:EXTRUDE
MOVL C00281 V=30.0 PL=1
CALL JOB:EXTRUDE
MOVL C00282 V=30.0 PL=1
CALL JOB:EXTRUDE
MOVL C00283 V=30.0 PL=1
CALL JOB:EXTRUDE
MOVL C00284 V=30.0 PL=1
CALL JOB:EXTRUDE
MOVL C00285 V=30.0 PL=1
CALL JOB:EXTRUDE
MOVL C00286 V=30.0 PL=1
CALL JOB:EXTRUDE
MOVL C00287 V=30.0 PL=1
CALL JOB:EXTRUDE
MOVL C00288 V=30.0 PL=1
CALL JOB:EXTRUDE
MOVL C00289 V=30.0 PL=1
CALL JOB:EXTRUDE
MOVL C00290 V=30.0 PL=1
CALL JOB:EXTRUDE
MOVL C00291 V=30.0 PL=1
CALL JOB:EXTRUDE
MOVL C00292 V=30.0 PL=1
CALL JOB:EXTRUDE
MOVL C00293 V=30.0 PL=1
CALL JOB:EXTRUDE
MOVL C00294 V=30.0 PL=1
CALL JOB:EXTRUDE
MOVL C00295 V=30.0 PL=1
CALL JOB:EXTRUDE
MOVL C00296 V=30.0 PL=1
CALL JOB:EXTRUDE
MOVL C00297 V=30.0 PL=1
CALL JOB:EXTRUDE
MOVL C00298 V=30.0 PL=1
CALL JOB:EXTRUDE
MOVL C00299 V=30.0 PL=1
CALL JOB:EXTRUDE
MOVL C00300 V=30.0 PL=1
CALL JOB:EXTRUDE
MOVL C00301 V=30.0 PL=1
CALL JOB:EXTRUDE
MOVL C00302 V=30.0 PL=1
CALL JOB:EXTRUDE
MOVL C00303 V=30.0 PL=1
CALL JOB:EXTRUDE
MOVL C00304 V=30.0 PL=1
CALL JOB:EXTRUDE
MOVL C00305 V=30.0 PL=1
CALL JOB:EXTRUDE
MOVL C00306 V=30.0 PL=1
CALL JOB:EXTRUDE
MOVL C00307 V=30.0 PL=1
CALL JOB:EXTRUDE
MOVL C00308 V=30.0 PL=1
CALL JOB:EXTRUDE
MOVL C00309 V=30.0 PL=1
CALL JOB:EXTRUDE
MOVL C00310 V=30.0 PL=1
CALL JOB:EXTRUDE
MOVL C00311 V=30.0 PL=1
CALL JOB:EXTRUDE
CALL JOB:EXTRUDE
MOVL C00312 V=130.0 PL=1
CALL JOB:EXTRUDE
CALL JOB:EXTRUDE
MOVL C00313 V=30.0 PL=1
CALL JOB:EXTRUDE
MOVL C00314 V=30.0 PL=1
CALL JOB:EXTRUDE
MOVL C00315 V=30.0 PL=1
CALL JOB:EXTRUDE
MOVL C00316 V=30.0 PL=1
CALL JOB:EXTRUDE
CALL JOB:EXTRUDE
MOVL C00317 V=130.0 PL=1
CALL JOB:EXTRUDE
CALL JOB:EXTRUDE
MOVL C00318 V=30.0 PL=1
CALL JOB:EXTRUDE
MOVL C00319 V=30.0 PL=1
CALL JOB:EXTRUDE
MOVL C00320 V=30.0 PL=1
CALL JOB:EXTRUDE
MOVL C00321 V=30.0 PL=1
CALL JOB:EXTRUDE
CALL JOB:EXTRUDE
MOVL C00322 V=130.0 PL=1
CALL JOB:EXTRUDE
CALL JOB:EXTRUDE
MOVL C00323 V=30.0 PL=1
CALL JOB:EXTRUDE
MOVL C00324 V=30.0 PL=1
CALL JOB:EXTRUDE
MOVL C00325 V=30.0 PL=1
CALL JOB:EXTRUDE
MOVL C00326 V=30.0 PL=1
CALL JOB:EXTRUDE
MOVL C00327 V=30.0 PL=1
CALL JOB:EXTRUDE
MOVL C00328 V=30.0 PL=1
CALL JOB:EXTRUDE
MOVL C00329 V=30.0 PL=1
CALL JOB:EXTRUDE
MOVL C00330 V=30.0 PL=1
CALL JOB:EXTRUDE
MOVL C00331 V=30.0 PL=1
CALL JOB:EXTRUDE
MOVL C00332 V=30.0 PL=1
CALL JOB:EXTRUDE
MOVL C00333 V=30.0 PL=1
CALL JOB:EXTRUDE
MOVL C00334 V=30.0 PL=1
CALL JOB:EXTRUDE
MOVL C00335 V=30.0 PL=1
CALL JOB:EXTRUDE
MOVL C00336 V=30.0 PL=1
CALL JOB:EXTRUDE
MOVL C00337 V=30.0 PL=1
CALL JOB:EXTRUDE
MOVL C00338 V=30.0 PL=1
CALL JOB:EXTRUDE
MOVL C00339 V=30.0 PL=1
CALL JOB:EXTRUDE
MOVL C00340 V=30.0 PL=1
CALL JOB:EXTRUDE
MOVL C00341 V=30.0 PL=1
CALL JOB:EXTRUDE
MOVL C00342 V=30.0 PL=1
CALL JOB:EXTRUDE
MOVL C00343 V=30.0 PL=1
CALL JOB:EXTRUDE
MOVL C00344 V=30.0 PL=1
CALL JOB:EXTRUDE
MOVL C00345 V=30.0 PL=1
CALL JOB:EXTRUDE
MOVL C00346 V=30.0 PL=1
CALL JOB:EXTRUDE
MOVL C00347 V=30.0 PL=1
CALL JOB:EXTRUDE
MOVL C00348 V=30.0 PL=1
CALL JOB:EXTRUDE
MOVL C00349 V=30.0 PL=1
CALL JOB:EXTRUDE
MOVL C00350 V=30.0 PL=1
CALL JOB:EXTRUDE
MOVL C00351 V=30.0 PL=1
CALL JOB:EXTRUDE
MOVL C00352 V=30.0 PL=1
CALL JOB:EXTRUDE
MOVL C00353 V=30.0 PL=1
CALL JOB:EXTRUDE
MOVL C00354 V=30.0 PL=1
CALL JOB:EXTRUDE
MOVL C00355 V=30.0 PL=1
CALL JOB:EXTRUDE
MOVL C00356 V=30.0 PL=1
CALL JOB:EXTRUDE
MOVL C00357 V=30.0 PL=1
CALL JOB:EXTRUDE
MOVL C00358 V=30.0 PL=1
CALL JOB:EXTRUDE
MOVL C00359 V=30.0 PL=1
CALL JOB:EXTRUDE
MOVL C00360 V=30.0 PL=1
CALL JOB:EXTRUDE
MOVL C00361 V=30.0 PL=1
CALL JOB:EXTRUDE
MOVL C00362 V=30.0 PL=1
CALL JOB:EXTRUDE
MOVL C00363 V=30.0 PL=1
CALL JOB:EXTRUDE
MOVL C00364 V=30.0 PL=1
CALL JOB:EXTRUDE
MOVL C00365 V=30.0 PL=1
CALL JOB:EXTRUDE
MOVL C00366 V=30.0 PL=1
CALL JOB:EXTRUDE
MOVL C00367 V=30.0 PL=1
CALL JOB:EXTRUDE
MOVL C00368 V=30.0 PL=1
CALL JOB:EXTRUDE
MOVL C00369 V=30.0 PL=1
CALL JOB:EXTRUDE
MOVL C00370 V=30.0 PL=1
CALL JOB:EXTRUDE
MOVL C00371 V=30.0 PL=1
CALL JOB:EXTRUDE
MOVL C00372 V=30.0 PL=1
CALL JOB:EXTRUDE
MOVL C00373 V=30.0 PL=1
CALL JOB:EXTRUDE
MOVL C00374 V=30.0 PL=1
CALL JOB:EXTRUDE
MOVL C00375 V=30.0 PL=1
CALL JOB:EXTRUDE
MOVL C00376 V=30.0 PL=1
CALL JOB:EXTRUDE
MOVL C00377 V=30.0 PL=1
CALL JOB:EXTRUDE
MOVL C00378 V=30.0 PL=1
CALL JOB:EXTRUDE
MOVL C00379 V=30.0 PL=1
CALL JOB:EXTRUDE
MOVL C00380 V=30.0 PL=1
CALL JOB:EXTRUDE
MOVL C00381 V=30.0 PL=1
CALL JOB:EXTRUDE
MOVL C00382 V=30.0 PL=1
CALL JOB:EXTRUDE
MOVL C00383 V=30.0 PL=1
CALL JOB:EXTRUDE
MOVL C00384 V=30.0 PL=1
CALL JOB:EXTRUDE
MOVL C00385 V=30.0 PL=1
CALL JOB:EXTRUDE
MOVL C00386 V=30.0 PL=1
CALL JOB:EXTRUDE
MOVL C00387 V=30.0 PL=1
CALL JOB:EXTRUDE
MOVL C00388 V=30.0 PL=1
CALL JOB:EXTRUDE
MOVL C00389 V=30.0 PL=1
CALL JOB:EXTRUDE
MOVL C00390 V=30.0 PL=1
CALL JOB:EXTRUDE
MOVL C00391 V=30.0 PL=1
CALL JOB:EXTRUDE
MOVL C00392 V=30.0 PL=1
CALL JOB:EXTRUDE
MOVL C00393 V=30.0 PL=1
CALL JOB:EXTRUDE
MOVL C00394 V=30.0 PL=1
CALL JOB:EXTRUDE
MOVL C00395 V=30.0 PL=1
CALL JOB:EXTRUDE
MOVL C00396 V=30.0 PL=1
CALL JOB:EXTRUDE
MOVL C00397 V=30.0 PL=1
CALL JOB:EXTRUDE
MOVL C00398 V=30.0 PL=1
CALL JOB:EXTRUDE
MOVL C00399 V=30.0 PL=1
CALL JOB:EXTRUDE
MOVL C00400 V=30.0 PL=1
CALL JOB:EXTRUDE
MOVL C00401 V=30.0 PL=1
CALL JOB:EXTRUDE
MOVL C00402 V=30.0 PL=1
CALL JOB:EXTRUDE
MOVL C00403 V=30.0 PL=1
CALL JOB:EXTRUDE
MOVL C00404 V=30.0 PL=1
CALL JOB:EXTRUDE
MOVL C00405 V=30.0 PL=1
CALL JOB:EXTRUDE
MOVL C00406 V=30.0 PL=1
CALL JOB:EXTRUDE
MOVL C00407 V=30.0 PL=1
CALL JOB:EXTRUDE
MOVL C00408 V=30.0 PL=1
CALL JOB:EXTRUDE
MOVL C00409 V=30.0 PL=1
CALL JOB:EXTRUDE
MOVL C00410 V=30.0 PL=1
CALL JOB:EXTRUDE
MOVL C00411 V=30.0 PL=1
CALL JOB:EXTRUDE
MOVL C00412 V=30.0 PL=1
CALL JOB:EXTRUDE
MOVL C00413 V=30.0 PL=1
CALL JOB:EXTRUDE
MOVL C00414 V=30.0 PL=1
CALL JOB:EXTRUDE
MOVL C00415 V=30.0 PL=1
CALL JOB:EXTRUDE
MOVL C00416 V=30.0 PL=1
CALL JOB:EXTRUDE
MOVL C00417 V=30.0 PL=1
CALL JOB:EXTRUDE
MOVL C00418 V=30.0 PL=1
CALL JOB:EXTRUDE
MOVL C00419 V=30.0 PL=1
CALL JOB:EXTRUDE
MOVL C00420 V=30.0 PL=1
CALL JOB:EXTRUDE
MOVL C00421 V=30.0 PL=1
CALL JOB:EXTRUDE
MOVL C00422 V=30.0 PL=1
CALL JOB:EXTRUDE
MOVL C00423 V=30.0 PL=1
CALL JOB:EXTRUDE
MOVL C00424 V=30.0 PL=1
CALL JOB:EXTRUDE
MOVL C00425 V=30.0 PL=1
CALL JOB:EXTRUDE
MOVL C00426 V=30.0 PL=1
CALL JOB:EXTRUDE
MOVL C00427 V=30.0 PL=1
CALL JOB:EXTRUDE
MOVL C00428 V=30.0 PL=1
CALL JOB:EXTRUDE
MOVL C00429 V=30.0 PL=1
CALL JOB:EXTRUDE
MOVL C00430 V=30.0 PL=1
CALL JOB:EXTRUDE
MOVL C00431 V=30.0 PL=1
CALL JOB:EXTRUDE
MOVL C00432 V=30.0 PL=1
CALL JOB:EXTRUDE
MOVL C00433 V=30.0 PL=1
CALL JOB:EXTRUDE
MOVL C00434 V=30.0 PL=1
CALL JOB:EXTRUDE
MOVL C00435 V=30.0 PL=1
CALL JOB:EXTRUDE
MOVL C00436 V=30.0 PL=1
CALL JOB:EXTRUDE
CALL JOB:EXTRUDE
MOVL C00437 V=130.0 PL=1
CALL JOB:EXTRUDE
CALL JOB:EXTRUDE
MOVL C00438 V=30.0 PL=1
CALL JOB:EXTRUDE
MOVL C00439 V=30.0 PL=1
CALL JOB:EXTRUDE
MOVL C00440 V=30.0 PL=1
CALL JOB:EXTRUDE
MOVL C00441 V=30.0 PL=1
CALL JOB:EXTRUDE
MOVL C00442 V=30.0 PL=1
CALL JOB:EXTRUDE
MOVL C00443 V=30.0 PL=1
CALL JOB:EXTRUDE
MOVL C00444 V=30.0 PL=1
CALL JOB:EXTRUDE
MOVL C00445 V=30.0 PL=1
CALL JOB:EXTRUDE
MOVL C00446 V=30.0 PL=1
CALL JOB:EXTRUDE
MOVL C00447 V=30.0 PL=1
CALL JOB:EXTRUDE
MOVL C00448 V=30.0 PL=1
CALL JOB:EXTRUDE
MOVL C00449 V=30.0 PL=1
CALL JOB:EXTRUDE
MOVL C00450 V=30.0 PL=1
CALL JOB:EXTRUDE
MOVL C00451 V=30.0 PL=1
CALL JOB:EXTRUDE
MOVL C00452 V=30.0 PL=1
CALL JOB:EXTRUDE
MOVL C00453 V=30.0 PL=1
CALL JOB:EXTRUDE
MOVL C00454 V=30.0 PL=1
CALL JOB:EXTRUDE
MOVL C00455 V=30.0 PL=1
CALL JOB:EXTRUDE
MOVL C00456 V=30.0 PL=1
CALL JOB:EXTRUDE
MOVL C00457 V=30.0 PL=1
CALL JOB:EXTRUDE
MOVL C00458 V=30.0 PL=1
CALL JOB:EXTRUDE
MOVL C00459 V=30.0 PL=1
CALL JOB:EXTRUDE
MOVL C00460 V=30.0 PL=1
CALL JOB:EXTRUDE
MOVL C00461 V=30.0 PL=1
CALL JOB:EXTRUDE
MOVL C00462 V=30.0 PL=1
CALL JOB:EXTRUDE
MOVL C00463 V=30.0 PL=1
CALL JOB:EXTRUDE
MOVL C00464 V=30.0 PL=1
CALL JOB:EXTRUDE
MOVL C00465 V=30.0 PL=1
CALL JOB:EXTRUDE
MOVL C00466 V=30.0 PL=1
CALL JOB:EXTRUDE
MOVL C00467 V=30.0 PL=1
CALL JOB:EXTRUDE
MOVL C00468 V=30.0 PL=1
CALL JOB:EXTRUDE
MOVL C00469 V=30.0 PL=1
MOVL C00470 V=130.0 PL=1
CALL JOB:EXTRUDE
MOVL C00471 V=30.0 PL=1
CALL JOB:EXTRUDE
MOVL C00472 V=30.0 PL=1
CALL JOB:EXTRUDE
MOVL C00473 V=30.0 PL=1
CALL JOB:EXTRUDE
MOVL C00474 V=30.0 PL=1
CALL JOB:EXTRUDE
MOVL C00475 V=30.0 PL=1
CALL JOB:EXTRUDE
MOVL C00476 V=30.0 PL=1
CALL JOB:EXTRUDE
MOVL C00477 V=30.0 PL=1
CALL JOB:EXTRUDE
MOVL C00478 V=30.0 PL=1
CALL JOB:EXTRUDE
MOVL C00479 V=30.0 PL=1
CALL JOB:EXTRUDE
MOVL C00480 V=30.0 PL=1
CALL JOB:EXTRUDE
MOVL C00481 V=30.0 PL=1
CALL JOB:EXTRUDE
MOVL C00482 V=30.0 PL=1
CALL JOB:EXTRUDE
MOVL C00483 V=30.0 PL=1
CALL JOB:EXTRUDE
MOVL C00484 V=30.0 PL=1
CALL JOB:EXTRUDE
MOVL C00485 V=30.0 PL=1
CALL JOB:EXTRUDE
MOVL C00486 V=30.0 PL=1
CALL JOB:EXTRUDE
MOVL C00487 V=30.0 PL=1
CALL JOB:EXTRUDE
MOVL C00488 V=30.0 PL=1
CALL JOB:EXTRUDE
MOVL C00489 V=30.0 PL=1
CALL JOB:EXTRUDE
MOVL C00490 V=30.0 PL=1
CALL JOB:EXTRUDE
MOVL C00491 V=30.0 PL=1
CALL JOB:EXTRUDE
MOVL C00492 V=30.0 PL=1
CALL JOB:EXTRUDE
MOVL C00493 V=30.0 PL=1
CALL JOB:EXTRUDE
MOVL C00494 V=30.0 PL=1
CALL JOB:EXTRUDE
MOVL C00495 V=30.0 PL=1
CALL JOB:EXTRUDE
MOVL C00496 V=30.0 PL=1
CALL JOB:EXTRUDE
MOVL C00497 V=30.0 PL=1
CALL JOB:EXTRUDE
MOVL C00498 V=30.0 PL=1
CALL JOB:EXTRUDE
MOVL C00499 V=30.0 PL=1
CALL JOB:EXTRUDE
MOVL C00500 V=30.0 PL=1
CALL JOB:EXTRUDE
MOVL C00501 V=30.0 PL=1
CALL JOB:EXTRUDE
MOVL C00502 V=30.0 PL=1
MOVL C00503 V=130.0 PL=1
CALL JOB:EXTRUDE
CALL JOB:EXTRUDE
MOVL C00504 V=130.0 PL=1
CALL JOB:EXTRUDE
CALL JOB:EXTRUDE
MOVL C00505 V=30.0 PL=1
CALL JOB:EXTRUDE
MOVL C00506 V=30.0 PL=1
CALL JOB:EXTRUDE
MOVL C00507 V=30.0 PL=1
CALL JOB:EXTRUDE
MOVL C00508 V=30.0 PL=1
CALL JOB:EXTRUDE
MOVL C00509 V=30.0 PL=1
CALL JOB:EXTRUDE
MOVL C00510 V=30.0 PL=1
CALL JOB:EXTRUDE
MOVL C00511 V=30.0 PL=1
CALL JOB:EXTRUDE
CALL JOB:EXTRUDE
MOVL C00512 V=130.0 PL=1
CALL JOB:EXTRUDE
CALL JOB:EXTRUDE
MOVL C00513 V=30.0 PL=1
CALL JOB:EXTRUDE
MOVL C00514 V=30.0 PL=1
CALL JOB:EXTRUDE
MOVL C00515 V=30.0 PL=1
CALL JOB:EXTRUDE
MOVL C00516 V=30.0 PL=1
MOVL C00517 V=130.0 PL=1
CALL JOB:EXTRUDE
MOVL C00518 V=30.0 PL=1
CALL JOB:EXTRUDE
MOVL C00519 V=30.0 PL=1
CALL JOB:EXTRUDE
MOVL C00520 V=30.0 PL=1
CALL JOB:EXTRUDE
MOVL C00521 V=30.0 PL=1
MOVL C00522 V=130.0 PL=1
CALL JOB:EXTRUDE
CALL JOB:EXTRUDE
MOVL C00523 V=130.0 PL=1
CALL JOB:EXTRUDE
CALL JOB:EXTRUDE
MOVL C00524 V=30.0 PL=1
MOVL C00525 V=130.0 PL=1
CALL JOB:EXTRUDE
MOVL C00526 V=30.0 PL=1
CALL JOB:EXTRUDE
MOVL C00527 V=30.0 PL=1
CALL JOB:EXTRUDE
MOVL C00528 V=30.0 PL=1
CALL JOB:EXTRUDE
MOVL C00529 V=30.0 PL=1
CALL JOB:EXTRUDE
MOVL C00530 V=30.0 PL=1
MOVL C00531 V=130.0 PL=1
CALL JOB:EXTRUDE
MOVL C00532 V=30.0 PL=1
MOVL C00533 V=130.0 PL=1
CALL JOB:EXTRUDE
MOVL C00534 V=30.0 PL=1
MOVL C00535 V=130.0 PL=1
CALL JOB:EXTRUDE
MOVL C00536 V=30.0 PL=1
CALL JOB:EXTRUDE
CALL JOB:EXTRUDE
MOVL C00537 V=130.0 PL=1
CALL JOB:EXTRUDE
CALL JOB:EXTRUDE
MOVL C00538 V=30.0 PL=1
CALL JOB:EXTRUDE
MOVL C00539 V=30.0 PL=1
CALL JOB:EXTRUDE
MOVL C00540 V=30.0 PL=1
CALL JOB:EXTRUDE
MOVL C00541 V=30.0 PL=1
CALL JOB:EXTRUDE
MOVL C00542 V=30.0 PL=1
CALL JOB:EXTRUDE
MOVL C00543 V=30.0 PL=1
CALL JOB:EXTRUDE
MOVL C00544 V=30.0 PL=1
CALL JOB:EXTRUDE
MOVL C00545 V=30.0 PL=1
CALL JOB:EXTRUDE
MOVL C00546 V=30.0 PL=1
CALL JOB:EXTRUDE
MOVL C00547 V=30.0 PL=1
CALL JOB:EXTRUDE
MOVL C00548 V=30.0 PL=1
CALL JOB:EXTRUDE
MOVL C00549 V=30.0 PL=1
CALL JOB:EXTRUDE
MOVL C00550 V=30.0 PL=1
CALL JOB:EXTRUDE
MOVL C00551 V=30.0 PL=1
CALL JOB:EXTRUDE
MOVL C00552 V=30.0 PL=1
CALL JOB:EXTRUDE
MOVL C00553 V=30.0 PL=1
CALL JOB:EXTRUDE
MOVL C00554 V=30.0 PL=1
CALL JOB:EXTRUDE
MOVL C00555 V=30.0 PL=1
CALL JOB:EXTRUDE
MOVL C00556 V=30.0 PL=1
CALL JOB:EXTRUDE
MOVL C00557 V=30.0 PL=1
CALL JOB:EXTRUDE
MOVL C00558 V=30.0 PL=1
CALL JOB:EXTRUDE
CALL JOB:EXTRUDE
MOVL C00559 V=130.0 PL=1
CALL JOB:EXTRUDE
CALL JOB:EXTRUDE
MOVL C00560 V=30.0 PL=1
CALL JOB:EXTRUDE
MOVL C00561 V=30.0 PL=1
CALL JOB:EXTRUDE
MOVL C00562 V=30.0 PL=1
CALL JOB:EXTRUDE
MOVL C00563 V=30.0 PL=1
CALL JOB:EXTRUDE
MOVL C00564 V=30.0 PL=1
CALL JOB:EXTRUDE
MOVL C00565 V=30.0 PL=1
CALL JOB:EXTRUDE
MOVL C00566 V=30.0 PL=1
CALL JOB:EXTRUDE
MOVL C00567 V=30.0 PL=1
CALL JOB:EXTRUDE
MOVL C00568 V=30.0 PL=1
CALL JOB:EXTRUDE
MOVL C00569 V=30.0 PL=1
CALL JOB:EXTRUDE
MOVL C00570 V=30.0 PL=1
CALL JOB:EXTRUDE
MOVL C00571 V=30.0 PL=1
CALL JOB:EXTRUDE
MOVL C00572 V=30.0 PL=1
CALL JOB:EXTRUDE
MOVL C00573 V=30.0 PL=1
CALL JOB:EXTRUDE
MOVL C00574 V=30.0 PL=1
CALL JOB:EXTRUDE
MOVL C00575 V=30.0 PL=1
CALL JOB:EXTRUDE
MOVL C00576 V=30.0 PL=1
CALL JOB:EXTRUDE
MOVL C00577 V=30.0 PL=1
CALL JOB:EXTRUDE
MOVL C00578 V=30.0 PL=1
CALL JOB:EXTRUDE
MOVL C00579 V=30.0 PL=1
CALL JOB:EXTRUDE
MOVL C00580 V=30.0 PL=1
CALL JOB:EXTRUDE
MOVL C00581 V=30.0 PL=1
CALL JOB:EXTRUDE
MOVL C00582 V=30.0 PL=1
CALL JOB:EXTRUDE
MOVL C00583 V=30.0 PL=1
CALL JOB:EXTRUDE
MOVL C00584 V=30.0 PL=1
CALL JOB:EXTRUDE
MOVL C00585 V=30.0 PL=1
CALL JOB:EXTRUDE
MOVL C00586 V=30.0 PL=1
CALL JOB:EXTRUDE
MOVL C00587 V=30.0 PL=1
CALL JOB:EXTRUDE
MOVL C00588 V=30.0 PL=1
CALL JOB:EXTRUDE
MOVL C00589 V=30.0 PL=1
CALL JOB:EXTRUDE
MOVL C00590 V=30.0 PL=1
CALL JOB:EXTRUDE
MOVL C00591 V=30.0 PL=1
CALL JOB:EXTRUDE
MOVL C00592 V=30.0 PL=1
CALL JOB:EXTRUDE
MOVL C00593 V=30.0 PL=1
CALL JOB:EXTRUDE
MOVL C00594 V=30.0 PL=1
CALL JOB:EXTRUDE
MOVL C00595 V=30.0 PL=1
CALL JOB:EXTRUDE
MOVL C00596 V=30.0 PL=1
CALL JOB:EXTRUDE
MOVL C00597 V=30.0 PL=1
CALL JOB:EXTRUDE
MOVL C00598 V=30.0 PL=1
CALL JOB:EXTRUDE
MOVL C00599 V=30.0 PL=1
CALL JOB:EXTRUDE
MOVL C00600 V=30.0 PL=1
CALL JOB:EXTRUDE
MOVL C00601 V=30.0 PL=1
CALL JOB:EXTRUDE
MOVL C00602 V=30.0 PL=1
CALL JOB:EXTRUDE
MOVL C00603 V=30.0 PL=1
CALL JOB:EXTRUDE
MOVL C00604 V=30.0 PL=1
CALL JOB:EXTRUDE
MOVL C00605 V=30.0 PL=1
CALL JOB:EXTRUDE
MOVL C00606 V=30.0 PL=1
CALL JOB:EXTRUDE
MOVL C00607 V=30.0 PL=1
CALL JOB:EXTRUDE
MOVL C00608 V=30.0 PL=1
CALL JOB:EXTRUDE
MOVL C00609 V=30.0 PL=1
CALL JOB:EXTRUDE
MOVL C00610 V=30.0 PL=1
CALL JOB:EXTRUDE
MOVL C00611 V=30.0 PL=1
CALL JOB:EXTRUDE
MOVL C00612 V=30.0 PL=1
CALL JOB:EXTRUDE
MOVL C00613 V=30.0 PL=1
CALL JOB:EXTRUDE
MOVL C00614 V=30.0 PL=1
CALL JOB:EXTRUDE
MOVL C00615 V=30.0 PL=1
CALL JOB:EXTRUDE
MOVL C00616 V=30.0 PL=1
CALL JOB:EXTRUDE
MOVL C00617 V=30.0 PL=1
CALL JOB:EXTRUDE
MOVL C00618 V=30.0 PL=1
CALL JOB:EXTRUDE
MOVL C00619 V=30.0 PL=1
CALL JOB:EXTRUDE
MOVL C00620 V=30.0 PL=1
CALL JOB:EXTRUDE
MOVL C00621 V=30.0 PL=1
CALL JOB:EXTRUDE
MOVL C00622 V=30.0 PL=1
CALL JOB:EXTRUDE
MOVL C00623 V=30.0 PL=1
CALL JOB:EXTRUDE
MOVL C00624 V=30.0 PL=1
CALL JOB:EXTRUDE
MOVL C00625 V=30.0 PL=1
CALL JOB:EXTRUDE
MOVL C00626 V=30.0 PL=1
CALL JOB:EXTRUDE
MOVL C00627 V=30.0 PL=1
CALL JOB:EXTRUDE
MOVL C00628 V=30.0 PL=1
CALL JOB:EXTRUDE
MOVL C00629 V=30.0 PL=1
CALL JOB:EXTRUDE
MOVL C00630 V=30.0 PL=1
CALL JOB:EXTRUDE
MOVL C00631 V=30.0 PL=1
CALL JOB:EXTRUDE
MOVL C00632 V=30.0 PL=1
CALL JOB:EXTRUDE
MOVL C00633 V=30.0 PL=1
CALL JOB:EXTRUDE
MOVL C00634 V=30.0 PL=1
CALL JOB:EXTRUDE
MOVL C00635 V=30.0 PL=1
CALL JOB:EXTRUDE
MOVL C00636 V=30.0 PL=1
CALL JOB:EXTRUDE
MOVL C00637 V=30.0 PL=1
CALL JOB:EXTRUDE
MOVL C00638 V=30.0 PL=1
CALL JOB:EXTRUDE
MOVL C00639 V=30.0 PL=1
CALL JOB:EXTRUDE
MOVL C00640 V=30.0 PL=1
CALL JOB:EXTRUDE
MOVL C00641 V=30.0 PL=1
CALL JOB:EXTRUDE
MOVL C00642 V=30.0 PL=1
CALL JOB:EXTRUDE
MOVL C00643 V=30.0 PL=1
CALL JOB:EXTRUDE
MOVL C00644 V=30.0 PL=1
CALL JOB:EXTRUDE
MOVL C00645 V=30.0 PL=1
CALL JOB:EXTRUDE
MOVL C00646 V=30.0 PL=1
CALL JOB:EXTRUDE
MOVL C00647 V=30.0 PL=1
CALL JOB:EXTRUDE
MOVL C00648 V=30.0 PL=1
CALL JOB:EXTRUDE
MOVL C00649 V=30.0 PL=1
CALL JOB:EXTRUDE
MOVL C00650 V=30.0 PL=1
CALL JOB:EXTRUDE
MOVL C00651 V=30.0 PL=1
CALL JOB:EXTRUDE
MOVL C00652 V=30.0 PL=1
CALL JOB:EXTRUDE
MOVL C00653 V=30.0 PL=1
CALL JOB:EXTRUDE
MOVL C00654 V=30.0 PL=1
CALL JOB:EXTRUDE
MOVL C00655 V=30.0 PL=1
CALL JOB:EXTRUDE
MOVL C00656 V=30.0 PL=1
CALL JOB:EXTRUDE
MOVL C00657 V=30.0 PL=1
CALL JOB:EXTRUDE
MOVL C00658 V=30.0 PL=1
CALL JOB:EXTRUDE
MOVL C00659 V=30.0 PL=1
CALL JOB:EXTRUDE
MOVL C00660 V=30.0 PL=1
CALL JOB:EXTRUDE
MOVL C00661 V=30.0 PL=1
CALL JOB:EXTRUDE
MOVL C00662 V=30.0 PL=1
CALL JOB:EXTRUDE
MOVL C00663 V=30.0 PL=1
CALL JOB:EXTRUDE
MOVL C00664 V=30.0 PL=1
CALL JOB:EXTRUDE
MOVL C00665 V=30.0 PL=1
CALL JOB:EXTRUDE
MOVL C00666 V=30.0 PL=1
CALL JOB:EXTRUDE
MOVL C00667 V=30.0 PL=1
CALL JOB:EXTRUDE
MOVL C00668 V=30.0 PL=1
CALL JOB:EXTRUDE
MOVL C00669 V=30.0 PL=1
CALL JOB:EXTRUDE
MOVL C00670 V=30.0 PL=1
CALL JOB:EXTRUDE
MOVL C00671 V=30.0 PL=1
CALL JOB:EXTRUDE
MOVL C00672 V=30.0 PL=1
CALL JOB:EXTRUDE
MOVL C00673 V=30.0 PL=1
CALL JOB:EXTRUDE
MOVL C00674 V=30.0 PL=1
CALL JOB:EXTRUDE
MOVL C00675 V=30.0 PL=1
CALL JOB:EXTRUDE
MOVL C00676 V=30.0 PL=1
CALL JOB:EXTRUDE
MOVL C00677 V=30.0 PL=1
CALL JOB:EXTRUDE
MOVL C00678 V=30.0 PL=1
CALL JOB:EXTRUDE
MOVL C00679 V=30.0 PL=1
CALL JOB:EXTRUDE
MOVL C00680 V=30.0 PL=1
CALL JOB:EXTRUDE
MOVL C00681 V=30.0 PL=1
CALL JOB:EXTRUDE
MOVL C00682 V=30.0 PL=1
CALL JOB:EXTRUDE
MOVL C00683 V=30.0 PL=1
CALL JOB:EXTRUDE
MOVL C00684 V=30.0 PL=1
CALL JOB:EXTRUDE
MOVL C00685 V=30.0 PL=1
CALL JOB:EXTRUDE
MOVL C00686 V=30.0 PL=1
CALL JOB:EXTRUDE
MOVL C00687 V=30.0 PL=1
CALL JOB:EXTRUDE
MOVL C00688 V=30.0 PL=1
CALL JOB:EXTRUDE
MOVL C00689 V=30.0 PL=1
CALL JOB:EXTRUDE
MOVL C00690 V=30.0 PL=1
CALL JOB:EXTRUDE
MOVL C00691 V=30.0 PL=1
CALL JOB:EXTRUDE
MOVL C00692 V=30.0 PL=1
CALL JOB:EXTRUDE
MOVL C00693 V=30.0 PL=1
CALL JOB:EXTRUDE
MOVL C00694 V=30.0 PL=1
CALL JOB:EXTRUDE
MOVL C00695 V=30.0 PL=1
CALL JOB:EXTRUDE
MOVL C00696 V=30.0 PL=1
CALL JOB:EXTRUDE
MOVL C00697 V=30.0 PL=1
CALL JOB:EXTRUDE
MOVL C00698 V=30.0 PL=1
CALL JOB:EXTRUDE
MOVL C00699 V=30.0 PL=1
CALL JOB:EXTRUDE
MOVL C00700 V=30.0 PL=1
CALL JOB:EXTRUDE
MOVL C00701 V=30.0 PL=1
CALL JOB:EXTRUDE
MOVL C00702 V=30.0 PL=1
CALL JOB:EXTRUDE
MOVL C00703 V=30.0 PL=1
CALL JOB:EXTRUDE
MOVL C00704 V=30.0 PL=1
CALL JOB:EXTRUDE
MOVL C00705 V=30.0 PL=1
CALL JOB:EXTRUDE
MOVL C00706 V=30.0 PL=1
CALL JOB:EXTRUDE
MOVL C00707 V=30.0 PL=1
CALL JOB:EXTRUDE
MOVL C00708 V=30.0 PL=1
CALL JOB:EXTRUDE
MOVL C00709 V=30.0 PL=1
CALL JOB:EXTRUDE
MOVL C00710 V=30.0 PL=1
CALL JOB:EXTRUDE
MOVL C00711 V=30.0 PL=1
CALL JOB:EXTRUDE
MOVL C00712 V=30.0 PL=1
CALL JOB:EXTRUDE
MOVL C00713 V=30.0 PL=1
CALL JOB:EXTRUDE
MOVL C00714 V=30.0 PL=1
CALL JOB:EXTRUDE
MOVL C00715 V=30.0 PL=1
CALL JOB:EXTRUDE
MOVL C00716 V=30.0 PL=1
CALL JOB:EXTRUDE
MOVL C00717 V=30.0 PL=1
CALL JOB:EXTRUDE
MOVL C00718 V=30.0 PL=1
CALL JOB:EXTRUDE
MOVL C00719 V=30.0 PL=1
CALL JOB:EXTRUDE
MOVL C00720 V=30.0 PL=1
CALL JOB:EXTRUDE
MOVL C00721 V=30.0 PL=1
CALL JOB:EXTRUDE
MOVL C00722 V=30.0 PL=1
CALL JOB:EXTRUDE
MOVL C00723 V=30.0 PL=1
CALL JOB:EXTRUDE
MOVL C00724 V=30.0 PL=1
CALL JOB:EXTRUDE
MOVL C00725 V=30.0 PL=1
CALL JOB:EXTRUDE
MOVL C00726 V=30.0 PL=1
CALL JOB:EXTRUDE
MOVL C00727 V=30.0 PL=1
CALL JOB:EXTRUDE
MOVL C00728 V=30.0 PL=1
CALL JOB:EXTRUDE
MOVL C00729 V=30.0 PL=1
CALL JOB:EXTRUDE
MOVL C00730 V=30.0 PL=1
CALL JOB:EXTRUDE
MOVL C00731 V=30.0 PL=1
CALL JOB:EXTRUDE
MOVL C00732 V=30.0 PL=1
CALL JOB:EXTRUDE
MOVL C00733 V=30.0 PL=1
CALL JOB:EXTRUDE
MOVL C00734 V=30.0 PL=1
CALL JOB:EXTRUDE
MOVL C00735 V=30.0 PL=1
CALL JOB:EXTRUDE
MOVL C00736 V=30.0 PL=1
CALL JOB:EXTRUDE
MOVL C00737 V=30.0 PL=1
CALL JOB:EXTRUDE
MOVL C00738 V=30.0 PL=1
CALL JOB:EXTRUDE
MOVL C00739 V=30.0 PL=1
CALL JOB:EXTRUDE
MOVL C00740 V=30.0 PL=1
CALL JOB:EXTRUDE
MOVL C00741 V=30.0 PL=1
CALL JOB:EXTRUDE
MOVL C00742 V=30.0 PL=1
CALL JOB:EXTRUDE
MOVL C00743 V=30.0 PL=1
CALL JOB:EXTRUDE
MOVL C00744 V=30.0 PL=1
CALL JOB:EXTRUDE
MOVL C00745 V=30.0 PL=1
CALL JOB:EXTRUDE
MOVL C00746 V=30.0 PL=1
CALL JOB:EXTRUDE
MOVL C00747 V=30.0 PL=1
CALL JOB:EXTRUDE
MOVL C00748 V=30.0 PL=1
CALL JOB:EXTRUDE
MOVL C00749 V=30.0 PL=1
CALL JOB:EXTRUDE
MOVL C00750 V=30.0 PL=1
CALL JOB:EXTRUDE
MOVL C00751 V=30.0 PL=1
CALL JOB:EXTRUDE
MOVL C00752 V=30.0 PL=1
CALL JOB:EXTRUDE
MOVL C00753 V=30.0 PL=1
CALL JOB:EXTRUDE
MOVL C00754 V=30.0 PL=1
CALL JOB:EXTRUDE
MOVL C00755 V=30.0 PL=1
CALL JOB:EXTRUDE
MOVL C00756 V=30.0 PL=1
CALL JOB:EXTRUDE
MOVL C00757 V=30.0 PL=1
CALL JOB:EXTRUDE
MOVL C00758 V=30.0 PL=1
CALL JOB:EXTRUDE
MOVL C00759 V=30.0 PL=1
CALL JOB:EXTRUDE
MOVL C00760 V=30.0 PL=1
CALL JOB:EXTRUDE
MOVL C00761 V=30.0 PL=1
CALL JOB:EXTRUDE
MOVL C00762 V=30.0 PL=1
CALL JOB:EXTRUDE
MOVL C00763 V=30.0 PL=1
CALL JOB:EXTRUDE
MOVL C00764 V=30.0 PL=1
CALL JOB:EXTRUDE
MOVL C00765 V=30.0 PL=1
CALL JOB:EXTRUDE
MOVL C00766 V=30.0 PL=1
CALL JOB:EXTRUDE
MOVL C00767 V=30.0 PL=1
CALL JOB:EXTRUDE
MOVL C00768 V=30.0 PL=1
CALL JOB:EXTRUDE
MOVL C00769 V=30.0 PL=1
CALL JOB:EXTRUDE
MOVL C00770 V=30.0 PL=1
CALL JOB:EXTRUDE
MOVL C00771 V=30.0 PL=1
CALL JOB:EXTRUDE
MOVL C00772 V=30.0 PL=1
CALL JOB:EXTRUDE
MOVL C00773 V=30.0 PL=1
CALL JOB:EXTRUDE
MOVL C00774 V=30.0 PL=1
CALL JOB:EXTRUDE
MOVL C00775 V=30.0 PL=1
CALL JOB:EXTRUDE
MOVL C00776 V=30.0 PL=1
CALL JOB:EXTRUDE
MOVL C00777 V=30.0 PL=1
CALL JOB:EXTRUDE
MOVL C00778 V=30.0 PL=1
CALL JOB:EXTRUDE
MOVL C00779 V=30.0 PL=1
CALL JOB:EXTRUDE
MOVL C00780 V=30.0 PL=1
CALL JOB:EXTRUDE
MOVL C00781 V=30.0 PL=1
CALL JOB:EXTRUDE
MOVL C00782 V=30.0 PL=1
CALL JOB:EXTRUDE
MOVL C00783 V=30.0 PL=1
CALL JOB:EXTRUDE
MOVL C00784 V=30.0 PL=1
CALL JOB:EXTRUDE
MOVL C00785 V=30.0 PL=1
CALL JOB:EXTRUDE
MOVL C00786 V=30.0 PL=1
CALL JOB:EXTRUDE
MOVL C00787 V=30.0 PL=1
CALL JOB:EXTRUDE
MOVL C00788 V=30.0 PL=1
CALL JOB:EXTRUDE
MOVL C00789 V=30.0 PL=1
CALL JOB:EXTRUDE
MOVL C00790 V=30.0 PL=1
CALL JOB:EXTRUDE
MOVL C00791 V=30.0 PL=1
CALL JOB:EXTRUDE
MOVL C00792 V=30.0 PL=1
CALL JOB:EXTRUDE
MOVL C00793 V=30.0 PL=1
CALL JOB:EXTRUDE
MOVL C00794 V=30.0 PL=1
CALL JOB:EXTRUDE
MOVL C00795 V=30.0 PL=1
CALL JOB:EXTRUDE
MOVL C00796 V=30.0 PL=1
CALL JOB:EXTRUDE
MOVL C00797 V=30.0 PL=1
CALL JOB:EXTRUDE
MOVL C00798 V=30.0 PL=1
CALL JOB:EXTRUDE
MOVL C00799 V=30.0 PL=1
CALL JOB:EXTRUDE
MOVL C00800 V=30.0 PL=1
CALL JOB:EXTRUDE
MOVL C00801 V=30.0 PL=1
CALL JOB:EXTRUDE
MOVL C00802 V=30.0 PL=1
CALL JOB:EXTRUDE
MOVL C00803 V=30.0 PL=1
CALL JOB:EXTRUDE
MOVL C00804 V=30.0 PL=1
CALL JOB:EXTRUDE
MOVL C00805 V=30.0 PL=1
CALL JOB:EXTRUDE
MOVL C00806 V=30.0 PL=1
CALL JOB:EXTRUDE
MOVL C00807 V=30.0 PL=1
CALL JOB:EXTRUDE
MOVL C00808 V=30.0 PL=1
CALL JOB:EXTRUDE
MOVL C00809 V=30.0 PL=1
CALL JOB:EXTRUDE
MOVL C00810 V=30.0 PL=1
CALL JOB:EXTRUDE
MOVL C00811 V=30.0 PL=1
CALL JOB:EXTRUDE
MOVL C00812 V=30.0 PL=1
CALL JOB:EXTRUDE
MOVL C00813 V=30.0 PL=1
CALL JOB:EXTRUDE
MOVL C00814 V=30.0 PL=1
CALL JOB:EXTRUDE
MOVL C00815 V=30.0 PL=1
CALL JOB:EXTRUDE
MOVL C00816 V=30.0 PL=1
CALL JOB:EXTRUDE
MOVL C00817 V=30.0 PL=1
CALL JOB:EXTRUDE
MOVL C00818 V=30.0 PL=1
CALL JOB:EXTRUDE
MOVL C00819 V=30.0 PL=1
CALL JOB:EXTRUDE
MOVL C00820 V=30.0 PL=1
CALL JOB:EXTRUDE
MOVL C00821 V=30.0 PL=1
CALL JOB:EXTRUDE
MOVL C00822 V=30.0 PL=1
CALL JOB:EXTRUDE
MOVL C00823 V=30.0 PL=1
CALL JOB:EXTRUDE
MOVL C00824 V=30.0 PL=1
CALL JOB:EXTRUDE
MOVL C00825 V=30.0 PL=1
CALL JOB:EXTRUDE
MOVL C00826 V=30.0 PL=1
CALL JOB:EXTRUDE
MOVL C00827 V=30.0 PL=1
CALL JOB:EXTRUDE
MOVL C00828 V=30.0 PL=1
CALL JOB:EXTRUDE
MOVL C00829 V=30.0 PL=1
CALL JOB:EXTRUDE
MOVL C00830 V=30.0 PL=1
CALL JOB:EXTRUDE
MOVL C00831 V=30.0 PL=1
CALL JOB:EXTRUDE
MOVL C00832 V=30.0 PL=1
CALL JOB:EXTRUDE
MOVL C00833 V=30.0 PL=1
CALL JOB:EXTRUDE
MOVL C00834 V=30.0 PL=1
CALL JOB:EXTRUDE
MOVL C00835 V=30.0 PL=1
CALL JOB:EXTRUDE
MOVL C00836 V=30.0 PL=1
CALL JOB:EXTRUDE
MOVL C00837 V=30.0 PL=1
CALL JOB:EXTRUDE
MOVL C00838 V=30.0 PL=1
CALL JOB:EXTRUDE
MOVL C00839 V=30.0 PL=1
CALL JOB:EXTRUDE
MOVL C00840 V=30.0 PL=1
CALL JOB:EXTRUDE
MOVL C00841 V=30.0 PL=1
CALL JOB:EXTRUDE
MOVL C00842 V=30.0 PL=1
CALL JOB:EXTRUDE
MOVL C00843 V=30.0 PL=1
CALL JOB:EXTRUDE
MOVL C00844 V=30.0 PL=1
CALL JOB:EXTRUDE
MOVL C00845 V=30.0 PL=1
CALL JOB:EXTRUDE
MOVL C00846 V=30.0 PL=1
CALL JOB:EXTRUDE
MOVL C00847 V=30.0 PL=1
CALL JOB:EXTRUDE
MOVL C00848 V=30.0 PL=1
CALL JOB:EXTRUDE
MOVL C00849 V=30.0 PL=1
CALL JOB:EXTRUDE
MOVL C00850 V=30.0 PL=1
CALL JOB:EXTRUDE
MOVL C00851 V=30.0 PL=1
CALL JOB:EXTRUDE
MOVL C00852 V=30.0 PL=1
CALL JOB:EXTRUDE
MOVL C00853 V=30.0 PL=1
CALL JOB:EXTRUDE
MOVL C00854 V=30.0 PL=1
CALL JOB:EXTRUDE
MOVL C00855 V=30.0 PL=1
CALL JOB:EXTRUDE
MOVL C00856 V=30.0 PL=1
CALL JOB:EXTRUDE
MOVL C00857 V=30.0 PL=1
CALL JOB:EXTRUDE
MOVL C00858 V=30.0 PL=1
CALL JOB:EXTRUDE
MOVL C00859 V=30.0 PL=1
CALL JOB:EXTRUDE
MOVL C00860 V=30.0 PL=1
CALL JOB:EXTRUDE
MOVL C00861 V=30.0 PL=1
CALL JOB:EXTRUDE
MOVL C00862 V=30.0 PL=1
CALL JOB:EXTRUDE
MOVL C00863 V=30.0 PL=1
CALL JOB:EXTRUDE
MOVL C00864 V=30.0 PL=1
CALL JOB:EXTRUDE
MOVL C00865 V=30.0 PL=1
CALL JOB:EXTRUDE
MOVL C00866 V=30.0 PL=1
CALL JOB:EXTRUDE
MOVL C00867 V=30.0 PL=1
CALL JOB:EXTRUDE
MOVL C00868 V=30.0 PL=1
CALL JOB:EXTRUDE
MOVL C00869 V=30.0 PL=1
CALL JOB:EXTRUDE
MOVL C00870 V=30.0 PL=1
CALL JOB:EXTRUDE
MOVL C00871 V=30.0 PL=1
CALL JOB:EXTRUDE
MOVL C00872 V=30.0 PL=1
CALL JOB:EXTRUDE
MOVL C00873 V=30.0 PL=1
CALL JOB:EXTRUDE
MOVL C00874 V=30.0 PL=1
CALL JOB:EXTRUDE
MOVL C00875 V=30.0 PL=1
CALL JOB:EXTRUDE
MOVL C00876 V=30.0 PL=1
CALL JOB:EXTRUDE
MOVL C00877 V=30.0 PL=1
CALL JOB:EXTRUDE
MOVL C00878 V=30.0 PL=1
CALL JOB:EXTRUDE
MOVL C00879 V=30.0 PL=1
CALL JOB:EXTRUDE
MOVL C00880 V=30.0 PL=1
CALL JOB:EXTRUDE
MOVL C00881 V=30.0 PL=1
CALL JOB:EXTRUDE
MOVL C00882 V=30.0 PL=1
CALL JOB:EXTRUDE
MOVL C00883 V=30.0 PL=1
CALL JOB:EXTRUDE
MOVL C00884 V=30.0 PL=1
CALL JOB:EXTRUDE
MOVL C00885 V=30.0 PL=1
CALL JOB:EXTRUDE
MOVL C00886 V=30.0 PL=1
CALL JOB:EXTRUDE
MOVL C00887 V=30.0 PL=1
CALL JOB:EXTRUDE
MOVL C00888 V=30.0 PL=1
CALL JOB:EXTRUDE
MOVL C00889 V=30.0 PL=1
CALL JOB:EXTRUDE
MOVL C00890 V=30.0 PL=1
CALL JOB:EXTRUDE
MOVL C00891 V=30.0 PL=1
CALL JOB:EXTRUDE
MOVL C00892 V=30.0 PL=1
CALL JOB:EXTRUDE
MOVL C00893 V=30.0 PL=1
CALL JOB:EXTRUDE
MOVL C00894 V=30.0 PL=1
CALL JOB:EXTRUDE
MOVL C00895 V=30.0 PL=1
CALL JOB:EXTRUDE
MOVL C00896 V=30.0 PL=1
CALL JOB:EXTRUDE
MOVL C00897 V=30.0 PL=1
CALL JOB:EXTRUDE
MOVL C00898 V=30.0 PL=1
CALL JOB:EXTRUDE
MOVL C00899 V=30.0 PL=1
CALL JOB:EXTRUDE
MOVL C00900 V=30.0 PL=1
CALL JOB:EXTRUDE
MOVL C00901 V=30.0 PL=1
CALL JOB:EXTRUDE
MOVL C00902 V=30.0 PL=1
CALL JOB:EXTRUDE
MOVL C00903 V=30.0 PL=1
CALL JOB:EXTRUDE
MOVL C00904 V=30.0 PL=1
CALL JOB:EXTRUDE
MOVL C00905 V=30.0 PL=1
CALL JOB:EXTRUDE
MOVL C00906 V=30.0 PL=1
CALL JOB:EXTRUDE
MOVL C00907 V=30.0 PL=1
CALL JOB:EXTRUDE
MOVL C00908 V=30.0 PL=1
CALL JOB:EXTRUDE
MOVL C00909 V=30.0 PL=1
CALL JOB:EXTRUDE
MOVL C00910 V=30.0 PL=1
CALL JOB:EXTRUDE
MOVL C00911 V=30.0 PL=1
CALL JOB:EXTRUDE
MOVL C00912 V=30.0 PL=1
CALL JOB:EXTRUDE
MOVL C00913 V=30.0 PL=1
CALL JOB:EXTRUDE
MOVL C00914 V=30.0 PL=1
CALL JOB:EXTRUDE
MOVL C00915 V=30.0 PL=1
CALL JOB:EXTRUDE
MOVL C00916 V=30.0 PL=1
CALL JOB:EXTRUDE
MOVL C00917 V=30.0 PL=1
CALL JOB:EXTRUDE
MOVL C00918 V=30.0 PL=1
CALL JOB:EXTRUDE
MOVL C00919 V=30.0 PL=1
CALL JOB:EXTRUDE
MOVL C00920 V=30.0 PL=1
CALL JOB:EXTRUDE
MOVL C00921 V=30.0 PL=1
CALL JOB:EXTRUDE
MOVL C00922 V=30.0 PL=1
CALL JOB:EXTRUDE
MOVL C00923 V=30.0 PL=1
CALL JOB:EXTRUDE
MOVL C00924 V=30.0 PL=1
CALL JOB:EXTRUDE
MOVL C00925 V=30.0 PL=1
CALL JOB:EXTRUDE
MOVL C00926 V=30.0 PL=1
CALL JOB:EXTRUDE
MOVL C00927 V=30.0 PL=1
CALL JOB:EXTRUDE
MOVL C00928 V=30.0 PL=1
CALL JOB:EXTRUDE
MOVL C00929 V=30.0 PL=1
CALL JOB:EXTRUDE
MOVL C00930 V=30.0 PL=1
CALL JOB:EXTRUDE
MOVL C00931 V=30.0 PL=1
CALL JOB:EXTRUDE
MOVL C00932 V=30.0 PL=1
CALL JOB:EXTRUDE
MOVL C00933 V=30.0 PL=1
CALL JOB:EXTRUDE
MOVL C00934 V=30.0 PL=1
CALL JOB:EXTRUDE
MOVL C00935 V=30.0 PL=1
CALL JOB:EXTRUDE
MOVL C00936 V=30.0 PL=1
CALL JOB:EXTRUDE
MOVL C00937 V=30.0 PL=1
CALL JOB:EXTRUDE
MOVL C00938 V=30.0 PL=1
CALL JOB:EXTRUDE
MOVL C00939 V=30.0 PL=1
CALL JOB:EXTRUDE
MOVL C00940 V=30.0 PL=1
CALL JOB:EXTRUDE
MOVL C00941 V=30.0 PL=1
CALL JOB:EXTRUDE
MOVL C00942 V=30.0 PL=1
CALL JOB:EXTRUDE
MOVL C00943 V=30.0 PL=1
CALL JOB:EXTRUDE
MOVL C00944 V=30.0 PL=1
CALL JOB:EXTRUDE
MOVL C00945 V=30.0 PL=1
CALL JOB:EXTRUDE
MOVL C00946 V=30.0 PL=1
CALL JOB:EXTRUDE
MOVL C00947 V=30.0 PL=1
CALL JOB:EXTRUDE
MOVL C00948 V=30.0 PL=1
CALL JOB:EXTRUDE
MOVL C00949 V=30.0 PL=1
CALL JOB:EXTRUDE
CALL JOB:EXTRUDE
MOVL C00950 V=130.0 PL=1
CALL JOB:EXTRUDE
CALL JOB:EXTRUDE
MOVL C00951 V=30.0 PL=1
CALL JOB:EXTRUDE
MOVL C00952 V=30.0 PL=1
CALL JOB:EXTRUDE
MOVL C00953 V=30.0 PL=1
CALL JOB:EXTRUDE
MOVL C00954 V=30.0 PL=1
CALL JOB:EXTRUDE
MOVL C00955 V=30.0 PL=1
CALL JOB:EXTRUDE
MOVL C00956 V=30.0 PL=1
CALL JOB:EXTRUDE
MOVL C00957 V=30.0 PL=1
CALL JOB:EXTRUDE
MOVL C00958 V=30.0 PL=1
CALL JOB:EXTRUDE
MOVL C00959 V=30.0 PL=1
CALL JOB:EXTRUDE
MOVL C00960 V=30.0 PL=1
CALL JOB:EXTRUDE
MOVL C00961 V=30.0 PL=1
CALL JOB:EXTRUDE
MOVL C00962 V=30.0 PL=1
CALL JOB:EXTRUDE
MOVL C00963 V=30.0 PL=1
CALL JOB:EXTRUDE
MOVL C00964 V=30.0 PL=1
CALL JOB:EXTRUDE
MOVL C00965 V=30.0 PL=1
CALL JOB:EXTRUDE
MOVL C00966 V=30.0 PL=1
CALL JOB:EXTRUDE
MOVL C00967 V=30.0 PL=1
CALL JOB:EXTRUDE
MOVL C00968 V=30.0 PL=1
CALL JOB:EXTRUDE
MOVL C00969 V=30.0 PL=1
CALL JOB:EXTRUDE
MOVL C00970 V=30.0 PL=1
CALL JOB:EXTRUDE
MOVL C00971 V=30.0 PL=1
CALL JOB:EXTRUDE
CALL JOB:EXTRUDE
MOVL C00972 V=130.0 PL=1
CALL JOB:EXTRUDE
CALL JOB:EXTRUDE
MOVL C00973 V=30.0 PL=1
CALL JOB:EXTRUDE
MOVL C00974 V=30.0 PL=1
CALL JOB:EXTRUDE
MOVL C00975 V=30.0 PL=1
CALL JOB:EXTRUDE
MOVL C00976 V=30.0 PL=1
MOVL C00977 V=130.0 PL=1
CALL JOB:EXTRUDE
MOVL C00978 V=30.0 PL=1
CALL JOB:EXTRUDE
MOVL C00979 V=30.0 PL=1
CALL JOB:EXTRUDE
MOVL C00980 V=30.0 PL=1
CALL JOB:EXTRUDE
END
